KUKA KRL program: ps_b_etb_res_c03_R.src, ps_b_etb_res_c03_R.dat

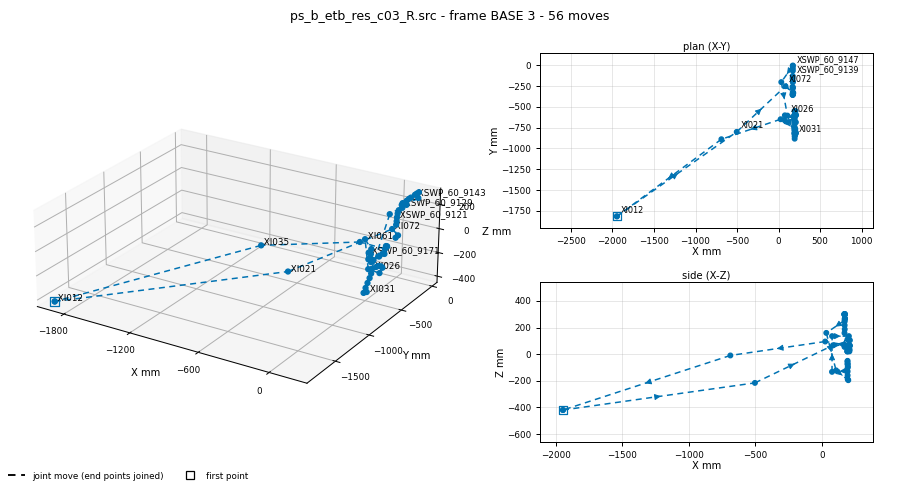
[picture p0: tool path of ps_b_etb_res_c03_R.src in frame BASE 3, 56 of 56 moves have a stored position in this frame; points joined in program order, loops and branches not executed]
--- ps_b_etb_res_c03_R.src ---
&ACCESS RVO2
&COMMENT Solda Atego STB
&PARAM DISKPATH = KRC:\R1\Program\olp
DEF ps_b_etb_res_c03_R( )
;FOLD INI
;FOLD SPOTTECH INI
USERSPOT(#INIT)
;ENDFOLD (SPOTTECH INI)
;FOLD GRIPPERTECH INI
USER_GRP(0,DUMMY,DUMMY,GDEFAULT)
;ENDFOLD (GRIPPERTECH INI)
  ;FOLD USER INI
    ;Make your modifications here

  ;ENDFOLD (USER INI)
;ENDFOLD (INI)

; Caraterizacao dos meios de producao
; Changes: Solda Respot - ATEGO STB
; Versao Atual: 30/03/2016
; Ferramenta: GUN C3
; Name: P13.050-R3
; optimised

chk_w5_wechs_ok ( )    ; CHECK GUN C3

if MaxStandMenge (3) then
 MaxStandmengeErreicht (3)
endif

IF (NOT(GHOST())) THEN
if Elektrodenwechsel ( 3 ) then
 e_fraes5 ()
endif
ENDIF

;FOLD PTP l012 Vel=100 % P_OLP37 Tool[5]:GUN C3 Base[3]:Atego/Axor;%{PE}%R 8.2.20,%MKUKATPBASIS,%CMOVE,%VPTP,%P 1:PTP, 2:l012, 3:, 5:100, 7:P_OLP37
$BWDSTART=FALSE
PDAT_ACT=PP_OLP37
FDAT_ACT=Fl012
BAS(#PTP_PARAMS,100)
PTP Xl012
;ENDFOLD

; AGUARDA LIBERACAO PARA SOLDAR RESPOT
;FOLD OUT 3333 'R3 trabalho concluído' State=FALSE ;%{PE}%R 8.2.20,%MKUKATPBASIS,%COUT,%VOUTX,%P 2:3333, 3:R3 trabalho concluído, 5:FALSE, 6:
$OUT[3333]=FALSE
;ENDFOLD
;FOLD OUT 3380 'Lib. p/ soldar Res Axor/Atego' State=TRUE ;%{PE}%R 8.2.20,%MKUKATPBASIS,%COUT,%VOUTX,%P 2:3380, 3:Lib. p/ soldar Res Axor/Atego, 5:TRUE, 6:
$OUT[3380]=TRUE
;ENDFOLD
;FOLD WAIT FOR ( IN 3380 'Lib. p/ soldar Res Axor/Atego' );%{PE}%R 8.2.20,%MKUKATPBASIS,%CEXT_WAIT_FOR,%VEXT_WAIT_FOR,%P 2:, 4:, 5:$IN, 6:3380, 7:Lib. p/ soldar Res Axor/Atego, 9:
WAIT FOR  ( $IN[3380] )
;ENDFOLD
;FOLD OUT 3380 'Lib. p/ soldar Res Axor/Atego' State=FALSE ;%{PE}%R 8.2.20,%MKUKATPBASIS,%COUT,%VOUTX,%P 2:3380, 3:Lib. p/ soldar Res Axor/Atego, 5:FALSE, 6:
$OUT[3380]=FALSE
;ENDFOLD
;FOLD OUT 3348 'Fora area GEOBOX' State=FALSE ;%{PE}%R 8.2.20,%MKUKATPBASIS,%COUT,%VOUTX,%P 2:3348, 3:Fora area GEOBOX, 5:FALSE, 6:
$OUT[3348]=FALSE
;ENDFOLD

;FOLD ; LIGA INTERTRAVAMENTO 4 SEGURANCA C/ GARRA DO R4;%{PE}%R 8.2.20,%MKUKATPBASIS,%CCOMMENT,%VNORMAL,%P 2:LIGA INTERTRAVAMENTO 4 SEGURANCA C/ GARRA DO R4
;ENDFOLD
;FOLD Collision.Monitoring_4_On ;%{PE}%MKUKATPUSER
COLLSTOP( 4, 1 ) ;Interrupt-Controlled
;ENDFOLD

;FOLD ; LIGA INTERTRAVAMENTO 13 COM R4 NA SOLDA;%{PE}%R 8.2.20,%MKUKATPBASIS,%CCOMMENT,%VNORMAL,%P 2:LIGA  INTERTRAVAMENTO  13  COM  R4  NA  SOLDA
;ENDFOLD
;FOLD Collision.Monitoring_AREA_7_On ;%{PE}%MKUKATPUSER
COLLSTOP( 13, 1 ) ;not Interrupt-Controlled
;ENDFOLD

;FOLD PTP l021 CONT Vel=100 % large Tool[5]:GUN C3 Base[3]:Atego/Axor;%{PE}%R 8.2.20,%MKUKATPBASIS,%CMOVE,%VPTP,%P 1:PTP, 2:l021, 3:C_DIS, 5:100, 7:large
$BWDSTART=FALSE
PDAT_ACT=Plarge
FDAT_ACT=Fl021
BAS(#PTP_PARAMS,100)
PTP Xl021 C_DIS
;ENDFOLD
;FOLD PTP l072 CONT Vel=100 % small Tool[5]:GUN C3 Base[3]:Atego/Axor;%{PE}%R 8.2.20,%MKUKATPBASIS,%CMOVE,%VPTP,%P 1:PTP, 2:l072, 3:C_DIS, 5:100, 7:small
$BWDSTART=FALSE
PDAT_ACT=Psmall
FDAT_ACT=Fl072
BAS(#PTP_PARAMS,100)
PTP Xl072 C_DIS
;ENDFOLD
;FOLD PTP l076 CONT Vel=100 % fin Tool[5]:GUN C3 Base[3]:Atego/Axor;%{PE}%R 8.2.20,%MKUKATPBASIS,%CMOVE,%VPTP,%P 1:PTP, 2:l076, 3:C_DIS, 5:100, 7:fin
$BWDSTART=FALSE
PDAT_ACT=Pfin
FDAT_ACT=Fl076
BAS(#PTP_PARAMS,100)
PTP Xl076 C_DIS
;ENDFOLD

;FOLD ; SWP_60_9103;%{PE}%R 8.2.20,%MKUKATPBASIS,%CCOMMENT,%VNORMAL,%P 2:SWP_60_9103
;ENDFOLD
;FOLD PTP SWP_60_9103 vmax SPOT Gun=3 RETR CLS PgNo1=200 ACTIVE=1 Tool[5]:GUN C3 Base[3]:Atego/Axor;%{PE}%R 8.2.2,%MKUKATPSPOT,%CSPOT,%VPTP,%P 1:PTP, 2:SWP_60_9103, 3:, 5:100, 7:vmax, 10:3, 12:#FIRST, 14:#CLO, 16:200, 18:1, 20:0, 22:0, 24:1, 25:NORMAL
$BWDSTART=FALSE
PDAT_ACT=Pvmax
FDAT_ACT=FSWP_60_9103
BAS(#PTP_PARAMS,Pvmax.VEL)
S_ACT.GUN=3
S_ACT.PAIR=SDEFAULT.PAIR
S_ACT.RETR=#CLO
S_ACT.CLO_TM=1
S_ACT.PGNO1=200
S_ACT.PGNO2=SDEFAULT.PGNO2
S_ACT.PRESS1=SDEFAULT.PRESS1
S_ACT.PRESS2=SDEFAULT.PRESS2
S_READY=FALSE
PTP XSWP_60_9103
USERSPOT(#SPOT, S_ACT)
WAIT FOR S_READY
;ENDFOLD

;FOLD ; SWP_60_9117;%{PE}%R 8.2.20,%MKUKATPBASIS,%CCOMMENT,%VNORMAL,%P 2:SWP_60_9117
;ENDFOLD
;FOLD PTP SWP_60_9117 vmax SPOT Gun=3 RETR CLS PgNo1=196 ACTIVE=1 Tool[5]:GUN C3 Base[3]:Atego/Axor;%{PE}%R 8.2.2,%MKUKATPSPOT,%CSPOT,%VPTP,%P 1:PTP, 2:SWP_60_9117, 3:, 5:100, 7:vmax, 10:3, 12:#FIRST, 14:#CLO, 16:196, 18:1, 20:0, 22:0, 24:1, 25:NORMAL
$BWDSTART=FALSE
PDAT_ACT=Pvmax
FDAT_ACT=FSWP_60_9117
BAS(#PTP_PARAMS,Pvmax.VEL)
S_ACT.GUN=3
S_ACT.PAIR=SDEFAULT.PAIR
S_ACT.RETR=#CLO
S_ACT.CLO_TM=1
S_ACT.PGNO1=196
S_ACT.PGNO2=SDEFAULT.PGNO2
S_ACT.PRESS1=SDEFAULT.PRESS1
S_ACT.PRESS2=SDEFAULT.PRESS2
S_READY=FALSE
PTP XSWP_60_9117
USERSPOT(#SPOT, S_ACT)
WAIT FOR S_READY
;ENDFOLD

;FOLD ; SWP_60_9119;%{PE}%R 8.2.20,%MKUKATPBASIS,%CCOMMENT,%VNORMAL,%P 2:SWP_60_9119
;ENDFOLD
;FOLD PTP SWP_60_9119 vmax SPOT Gun=3 RETR CLS PgNo1=196 ACTIVE=1 Tool[5]:GUN C3 Base[3]:Atego/Axor;%{PE}%R 8.2.2,%MKUKATPSPOT,%CSPOT,%VPTP,%P 1:PTP, 2:SWP_60_9119, 3:, 5:100, 7:vmax, 10:3, 12:#FIRST, 14:#CLO, 16:196, 18:1, 20:0, 22:0, 24:1, 25:NORMAL
$BWDSTART=FALSE
PDAT_ACT=Pvmax
FDAT_ACT=FSWP_60_9119
BAS(#PTP_PARAMS,Pvmax.VEL)
S_ACT.GUN=3
S_ACT.PAIR=SDEFAULT.PAIR
S_ACT.RETR=#CLO
S_ACT.CLO_TM=1
S_ACT.PGNO1=196
S_ACT.PGNO2=SDEFAULT.PGNO2
S_ACT.PRESS1=SDEFAULT.PRESS1
S_ACT.PRESS2=SDEFAULT.PRESS2
S_READY=FALSE
PTP XSWP_60_9119
USERSPOT(#SPOT, S_ACT)
WAIT FOR S_READY
;ENDFOLD

;FOLD ; SWP_60_9121;%{PE}%R 8.2.20,%MKUKATPBASIS,%CCOMMENT,%VNORMAL,%P 2:SWP_60_9121
;ENDFOLD
;FOLD PTP SWP_60_9121 vmax SPOT Gun=3 RETR CLS PgNo1=196 ACTIVE=1 Tool[5]:GUN C3 Base[3]:Atego/Axor;%{PE}%R 8.2.2,%MKUKATPSPOT,%CSPOT,%VPTP,%P 1:PTP, 2:SWP_60_9121, 3:, 5:100, 7:vmax, 10:3, 12:#FIRST, 14:#CLO, 16:196, 18:1, 20:0, 22:0, 24:1, 25:NORMAL
$BWDSTART=FALSE
PDAT_ACT=Pvmax
FDAT_ACT=FSWP_60_9121
BAS(#PTP_PARAMS,Pvmax.VEL)
S_ACT.GUN=3
S_ACT.PAIR=SDEFAULT.PAIR
S_ACT.RETR=#CLO
S_ACT.CLO_TM=1
S_ACT.PGNO1=196
S_ACT.PGNO2=SDEFAULT.PGNO2
S_ACT.PRESS1=SDEFAULT.PRESS1
S_ACT.PRESS2=SDEFAULT.PRESS2
S_READY=FALSE
PTP XSWP_60_9121
USERSPOT(#SPOT, S_ACT)
WAIT FOR S_READY
;ENDFOLD

;FOLD ; SWP_60_9123;%{PE}%R 8.2.20,%MKUKATPBASIS,%CCOMMENT,%VNORMAL,%P 2:SWP_60_9123
;ENDFOLD
;FOLD PTP SWP_60_9123 vmax SPOT Gun=3 RETR CLS PgNo1=196 ACTIVE=1 Tool[5]:GUN C3 Base[3]:Atego/Axor;%{PE}%R 8.2.2,%MKUKATPSPOT,%CSPOT,%VPTP,%P 1:PTP, 2:SWP_60_9123, 3:, 5:100, 7:vmax, 10:3, 12:#FIRST, 14:#CLO, 16:196, 18:1, 20:0, 22:0, 24:1, 25:NORMAL
$BWDSTART=FALSE
PDAT_ACT=Pvmax
FDAT_ACT=FSWP_60_9123
BAS(#PTP_PARAMS,Pvmax.VEL)
S_ACT.GUN=3
S_ACT.PAIR=SDEFAULT.PAIR
S_ACT.RETR=#CLO
S_ACT.CLO_TM=1
S_ACT.PGNO1=196
S_ACT.PGNO2=SDEFAULT.PGNO2
S_ACT.PRESS1=SDEFAULT.PRESS1
S_ACT.PRESS2=SDEFAULT.PRESS2
S_READY=FALSE
PTP XSWP_60_9123
USERSPOT(#SPOT, S_ACT)
WAIT FOR S_READY
;ENDFOLD

;FOLD ; SWP_60_9125;%{PE}%R 8.2.20,%MKUKATPBASIS,%CCOMMENT,%VNORMAL,%P 2:SWP_60_9125
;ENDFOLD
;FOLD PTP SWP_60_9125 vmax SPOT Gun=3 RETR CLS PgNo1=196 ACTIVE=1 Tool[5]:GUN C3 Base[3]:Atego/Axor;%{PE}%R 8.2.2,%MKUKATPSPOT,%CSPOT,%VPTP,%P 1:PTP, 2:SWP_60_9125, 3:, 5:100, 7:vmax, 10:3, 12:#FIRST, 14:#CLO, 16:196, 18:1, 20:0, 22:0, 24:1, 25:NORMAL
$BWDSTART=FALSE
PDAT_ACT=Pvmax
FDAT_ACT=FSWP_60_9125
BAS(#PTP_PARAMS,Pvmax.VEL)
S_ACT.GUN=3
S_ACT.PAIR=SDEFAULT.PAIR
S_ACT.RETR=#CLO
S_ACT.CLO_TM=1
S_ACT.PGNO1=196
S_ACT.PGNO2=SDEFAULT.PGNO2
S_ACT.PRESS1=SDEFAULT.PRESS1
S_ACT.PRESS2=SDEFAULT.PRESS2
S_READY=FALSE
PTP XSWP_60_9125
USERSPOT(#SPOT, S_ACT)
WAIT FOR S_READY
;ENDFOLD

;FOLD ; SWP_60_9129;%{PE}%R 8.2.20,%MKUKATPBASIS,%CCOMMENT,%VNORMAL,%P 2:SWP_60_9129
;ENDFOLD
;FOLD PTP SWP_60_9129 vmax SPOT Gun=3 RETR CLS PgNo1=196 ACTIVE=1 Tool[5]:GUN C3 Base[3]:Atego/Axor;%{PE}%R 8.2.2,%MKUKATPSPOT,%CSPOT,%VPTP,%P 1:PTP, 2:SWP_60_9129, 3:, 5:100, 7:vmax, 10:3, 12:#FIRST, 14:#CLO, 16:196, 18:1, 20:0, 22:0, 24:1, 25:NORMAL
$BWDSTART=FALSE
PDAT_ACT=Pvmax
FDAT_ACT=FSWP_60_9129
BAS(#PTP_PARAMS,Pvmax.VEL)
S_ACT.GUN=3
S_ACT.PAIR=SDEFAULT.PAIR
S_ACT.RETR=#CLO
S_ACT.CLO_TM=1
S_ACT.PGNO1=196
S_ACT.PGNO2=SDEFAULT.PGNO2
S_ACT.PRESS1=SDEFAULT.PRESS1
S_ACT.PRESS2=SDEFAULT.PRESS2
S_READY=FALSE
PTP XSWP_60_9129
USERSPOT(#SPOT, S_ACT)
WAIT FOR S_READY
;ENDFOLD

;FOLD ; SWP_60_9131;%{PE}%R 8.2.20,%MKUKATPBASIS,%CCOMMENT,%VNORMAL,%P 2:SWP_60_9131
;ENDFOLD
;FOLD PTP SWP_60_9131 vmax SPOT Gun=3 RETR CLS PgNo1=196 ACTIVE=1 Tool[5]:GUN C3 Base[3]:Atego/Axor;%{PE}%R 8.2.2,%MKUKATPSPOT,%CSPOT,%VPTP,%P 1:PTP, 2:SWP_60_9131, 3:, 5:100, 7:vmax, 10:3, 12:#FIRST, 14:#CLO, 16:196, 18:1, 20:0, 22:0, 24:1, 25:NORMAL
$BWDSTART=FALSE
PDAT_ACT=Pvmax
FDAT_ACT=FSWP_60_9131
BAS(#PTP_PARAMS,Pvmax.VEL)
S_ACT.GUN=3
S_ACT.PAIR=SDEFAULT.PAIR
S_ACT.RETR=#CLO
S_ACT.CLO_TM=1
S_ACT.PGNO1=196
S_ACT.PGNO2=SDEFAULT.PGNO2
S_ACT.PRESS1=SDEFAULT.PRESS1
S_ACT.PRESS2=SDEFAULT.PRESS2
S_READY=FALSE
PTP XSWP_60_9131
USERSPOT(#SPOT, S_ACT)
WAIT FOR S_READY
;ENDFOLD

;FOLD PTP l077 CONT Vel=100 % fin Tool[5]:GUN C3 Base[3]:Atego/Axor;%{PE}%R 8.2.20,%MKUKATPBASIS,%CMOVE,%VPTP,%P 1:PTP, 2:l077, 3:C_DIS, 5:100, 7:fin
$BWDSTART=FALSE
PDAT_ACT=Pfin
FDAT_ACT=Fl077
BAS(#PTP_PARAMS,100)
PTP Xl077 C_DIS
;ENDFOLD
;FOLD PTP l078 CONT Vel=100 % fin Tool[5]:GUN C3 Base[3]:Atego/Axor;%{PE}%R 8.2.20,%MKUKATPBASIS,%CMOVE,%VPTP,%P 1:PTP, 2:l078, 3:C_DIS, 5:100, 7:fin
$BWDSTART=FALSE
PDAT_ACT=Pfin
FDAT_ACT=Fl078
BAS(#PTP_PARAMS,100)
PTP Xl078 C_DIS
;ENDFOLD

;FOLD ; SWP_60_9135;%{PE}%R 8.2.20,%MKUKATPBASIS,%CCOMMENT,%VNORMAL,%P 2:SWP_60_9135
;ENDFOLD
;FOLD PTP SWP_60_9135 vmax SPOT Gun=3 RETR CLS PgNo1=196 ACTIVE=1 Tool[5]:GUN C3 Base[3]:Atego/Axor;%{PE}%R 8.2.2,%MKUKATPSPOT,%CSPOT,%VPTP,%P 1:PTP, 2:SWP_60_9135, 3:, 5:100, 7:vmax, 10:3, 12:#FIRST, 14:#CLO, 16:196, 18:1, 20:0, 22:0, 24:1, 25:NORMAL
$BWDSTART=FALSE
PDAT_ACT=Pvmax
FDAT_ACT=FSWP_60_9135
BAS(#PTP_PARAMS,Pvmax.VEL)
S_ACT.GUN=3
S_ACT.PAIR=SDEFAULT.PAIR
S_ACT.RETR=#CLO
S_ACT.CLO_TM=1
S_ACT.PGNO1=196
S_ACT.PGNO2=SDEFAULT.PGNO2
S_ACT.PRESS1=SDEFAULT.PRESS1
S_ACT.PRESS2=SDEFAULT.PRESS2
S_READY=FALSE
PTP XSWP_60_9135
USERSPOT(#SPOT, S_ACT)
WAIT FOR S_READY
;ENDFOLD

;FOLD ; SWP_60_9137;%{PE}%R 8.2.20,%MKUKATPBASIS,%CCOMMENT,%VNORMAL,%P 2:SWP_60_9137
;ENDFOLD
;FOLD PTP SWP_60_9137 vmax SPOT Gun=3 RETR CLS PgNo1=196 ACTIVE=1 Tool[5]:GUN C3 Base[3]:Atego/Axor;%{PE}%R 8.2.2,%MKUKATPSPOT,%CSPOT,%VPTP,%P 1:PTP, 2:SWP_60_9137, 3:, 5:100, 7:vmax, 10:3, 12:#FIRST, 14:#CLO, 16:196, 18:1, 20:0, 22:0, 24:1, 25:NORMAL
$BWDSTART=FALSE
PDAT_ACT=Pvmax
FDAT_ACT=FSWP_60_9137
BAS(#PTP_PARAMS,Pvmax.VEL)
S_ACT.GUN=3
S_ACT.PAIR=SDEFAULT.PAIR
S_ACT.RETR=#CLO
S_ACT.CLO_TM=1
S_ACT.PGNO1=196
S_ACT.PGNO2=SDEFAULT.PGNO2
S_ACT.PRESS1=SDEFAULT.PRESS1
S_ACT.PRESS2=SDEFAULT.PRESS2
S_READY=FALSE
PTP XSWP_60_9137
USERSPOT(#SPOT, S_ACT)
WAIT FOR S_READY
;ENDFOLD

;FOLD ; SWP_60_9139;%{PE}%R 8.2.20,%MKUKATPBASIS,%CCOMMENT,%VNORMAL,%P 2:SWP_60_9139
;ENDFOLD
;FOLD PTP SWP_60_9139 vmax SPOT Gun=3 RETR CLS PgNo1=196 ACTIVE=1 Tool[5]:GUN C3 Base[3]:Atego/Axor;%{PE}%R 8.2.2,%MKUKATPSPOT,%CSPOT,%VPTP,%P 1:PTP, 2:SWP_60_9139, 3:, 5:100, 7:vmax, 10:3, 12:#FIRST, 14:#CLO, 16:196, 18:1, 20:0, 22:0, 24:1, 25:NORMAL
$BWDSTART=FALSE
PDAT_ACT=Pvmax
FDAT_ACT=FSWP_60_9139
BAS(#PTP_PARAMS,Pvmax.VEL)
S_ACT.GUN=3
S_ACT.PAIR=SDEFAULT.PAIR
S_ACT.RETR=#CLO
S_ACT.CLO_TM=1
S_ACT.PGNO1=196
S_ACT.PGNO2=SDEFAULT.PGNO2
S_ACT.PRESS1=SDEFAULT.PRESS1
S_ACT.PRESS2=SDEFAULT.PRESS2
S_READY=FALSE
PTP XSWP_60_9139
USERSPOT(#SPOT, S_ACT)
WAIT FOR S_READY
;ENDFOLD

;FOLD ; SWP_60_9143;%{PE}%R 8.2.20,%MKUKATPBASIS,%CCOMMENT,%VNORMAL,%P 2:SWP_60_9143
;ENDFOLD
;FOLD PTP SWP_60_9143 vmax SPOT Gun=3 RETR CLS PgNo1=196 ACTIVE=1 Tool[5]:GUN C3 Base[3]:Atego/Axor;%{PE}%R 8.2.2,%MKUKATPSPOT,%CSPOT,%VPTP,%P 1:PTP, 2:SWP_60_9143, 3:, 5:100, 7:vmax, 10:3, 12:#FIRST, 14:#CLO, 16:196, 18:1, 20:0, 22:0, 24:1, 25:NORMAL
$BWDSTART=FALSE
PDAT_ACT=Pvmax
FDAT_ACT=FSWP_60_9143
BAS(#PTP_PARAMS,Pvmax.VEL)
S_ACT.GUN=3
S_ACT.PAIR=SDEFAULT.PAIR
S_ACT.RETR=#CLO
S_ACT.CLO_TM=1
S_ACT.PGNO1=196
S_ACT.PGNO2=SDEFAULT.PGNO2
S_ACT.PRESS1=SDEFAULT.PRESS1
S_ACT.PRESS2=SDEFAULT.PRESS2
S_READY=FALSE
PTP XSWP_60_9143
USERSPOT(#SPOT, S_ACT)
WAIT FOR S_READY
;ENDFOLD

;FOLD ; SWP_60_9145;%{PE}%R 8.2.20,%MKUKATPBASIS,%CCOMMENT,%VNORMAL,%P 2:SWP_60_9145
;ENDFOLD
;FOLD PTP SWP_60_9145 vmax SPOT Gun=3 RETR CLS PgNo1=196 ACTIVE=1 Tool[5]:GUN C3 Base[3]:Atego/Axor;%{PE}%R 8.2.2,%MKUKATPSPOT,%CSPOT,%VPTP,%P 1:PTP, 2:SWP_60_9145, 3:, 5:100, 7:vmax, 10:3, 12:#FIRST, 14:#CLO, 16:196, 18:1, 20:0, 22:0, 24:1, 25:NORMAL
$BWDSTART=FALSE
PDAT_ACT=Pvmax
FDAT_ACT=FSWP_60_9145
BAS(#PTP_PARAMS,Pvmax.VEL)
S_ACT.GUN=3
S_ACT.PAIR=SDEFAULT.PAIR
S_ACT.RETR=#CLO
S_ACT.CLO_TM=1
S_ACT.PGNO1=196
S_ACT.PGNO2=SDEFAULT.PGNO2
S_ACT.PRESS1=SDEFAULT.PRESS1
S_ACT.PRESS2=SDEFAULT.PRESS2
S_READY=FALSE
PTP XSWP_60_9145
USERSPOT(#SPOT, S_ACT)
WAIT FOR S_READY
;ENDFOLD

;FOLD ; SWP_60_9147;%{PE}%R 8.2.20,%MKUKATPBASIS,%CCOMMENT,%VNORMAL,%P 2:SWP_60_9147
;ENDFOLD
;FOLD PTP SWP_60_9147 vmax SPOT Gun=3 RETR CLS PgNo1=196 ACTIVE=1 Tool[5]:GUN C3 Base[3]:Atego/Axor;%{PE}%R 8.2.2,%MKUKATPSPOT,%CSPOT,%VPTP,%P 1:PTP, 2:SWP_60_9147, 3:, 5:100, 7:vmax, 10:3, 12:#FIRST, 14:#CLO, 16:196, 18:1, 20:0, 22:0, 24:1, 25:NORMAL
$BWDSTART=FALSE
PDAT_ACT=Pvmax
FDAT_ACT=FSWP_60_9147
BAS(#PTP_PARAMS,Pvmax.VEL)
S_ACT.GUN=3
S_ACT.PAIR=SDEFAULT.PAIR
S_ACT.RETR=#CLO
S_ACT.CLO_TM=1
S_ACT.PGNO1=196
S_ACT.PGNO2=SDEFAULT.PGNO2
S_ACT.PRESS1=SDEFAULT.PRESS1
S_ACT.PRESS2=SDEFAULT.PRESS2
S_READY=FALSE
PTP XSWP_60_9147
USERSPOT(#SPOT, S_ACT)
WAIT FOR S_READY
;ENDFOLD

;FOLD PTP l116 CONT Vel=100 % small Tool[5]:GUN C3 Base[3]:Atego/Axor;%{PE}%R 8.2.20,%MKUKATPBASIS,%CMOVE,%VPTP,%P 1:PTP, 2:l116, 3:C_DIS, 5:100, 7:small
$BWDSTART=FALSE
PDAT_ACT=Psmall
FDAT_ACT=Fl116
BAS(#PTP_PARAMS,100)
PTP Xl116 C_DIS
;ENDFOLD
;FOLD PTP l044 CONT Vel=100 % large Tool[5]:GUN C3 Base[3]:Atego/Axor;%{PE}%R 8.2.20,%MKUKATPBASIS,%CMOVE,%VPTP,%P 1:PTP, 2:l044, 3:C_DIS, 5:100, 7:large
$BWDSTART=FALSE
PDAT_ACT=Plarge
FDAT_ACT=Fl044
BAS(#PTP_PARAMS,100)
PTP Xl044 C_DIS
;ENDFOLD
;FOLD PTP l026 CONT Vel=100 % large Tool[5]:GUN C3 Base[3]:Atego/Axor;%{PE}%R 8.2.20,%MKUKATPBASIS,%CMOVE,%VPTP,%P 1:PTP, 2:l026, 3:C_DIS, 5:100, 7:large
$BWDSTART=FALSE
PDAT_ACT=Plarge
FDAT_ACT=Fl026
BAS(#PTP_PARAMS,100)
PTP Xl026 C_DIS
;ENDFOLD
;FOLD PTP l031 CONT Vel=100 % fin Tool[5]:GUN C3 Base[3]:Atego/Axor;%{PE}%R 8.2.20,%MKUKATPBASIS,%CMOVE,%VPTP,%P 1:PTP, 2:l031, 3:C_DIS, 5:100, 7:fin
$BWDSTART=FALSE
PDAT_ACT=Pfin
FDAT_ACT=Fl031
BAS(#PTP_PARAMS,100)
PTP Xl031 C_DIS
;ENDFOLD

;FOLD ; SWP_60_9041;%{PE}%R 8.2.20,%MKUKATPBASIS,%CCOMMENT,%VNORMAL,%P 2:SWP_60_9041
;ENDFOLD
;FOLD PTP SWP_60_9041 vmax SPOT Gun=3 RETR CLS PgNo1=196 ACTIVE=1 Tool[5]:GUN C3 Base[3]:Atego/Axor;%{PE}%R 8.2.2,%MKUKATPSPOT,%CSPOT,%VPTP,%P 1:PTP, 2:SWP_60_9041, 3:, 5:100, 7:vmax, 10:3, 12:#FIRST, 14:#CLO, 16:196, 18:1, 20:0, 22:0, 24:1, 25:NORMAL
$BWDSTART=FALSE
PDAT_ACT=Pvmax
FDAT_ACT=FSWP_60_9041
BAS(#PTP_PARAMS,Pvmax.VEL)
S_ACT.GUN=3
S_ACT.PAIR=SDEFAULT.PAIR
S_ACT.RETR=#CLO
S_ACT.CLO_TM=1
S_ACT.PGNO1=196
S_ACT.PGNO2=SDEFAULT.PGNO2
S_ACT.PRESS1=SDEFAULT.PRESS1
S_ACT.PRESS2=SDEFAULT.PRESS2
S_READY=FALSE
PTP XSWP_60_9041
USERSPOT(#SPOT, S_ACT)
WAIT FOR S_READY
;ENDFOLD

;FOLD ; DESLIGA INTERTRAVAMENTO 13 COM R4 NA SOLDA;%{PE}%R 8.2.20,%MKUKATPBASIS,%CCOMMENT,%VNORMAL,%P 2:DESLIGA  INTERTRAVAMENTO  13  COM  R4  NA  SOLDA
;ENDFOLD
;FOLD Collision.Monitoring_AREA_7_Off . ;%{PE}%MKUKATPUSER
COLLSTOP( 13, 2+0 )
;ENDFOLD

;FOLD ; SWP_60_9039;%{PE}%R 8.2.20,%MKUKATPBASIS,%CCOMMENT,%VNORMAL,%P 2:SWP_60_9039
;ENDFOLD
;FOLD PTP SWP_60_9039 vmax SPOT Gun=3 RETR CLS PgNo1=196 ACTIVE=1 Tool[5]:GUN C3 Base[3]:Atego/Axor;%{PE}%R 8.2.2,%MKUKATPSPOT,%CSPOT,%VPTP,%P 1:PTP, 2:SWP_60_9039, 3:, 5:100, 7:vmax, 10:3, 12:#FIRST, 14:#CLO, 16:196, 18:1, 20:0, 22:0, 24:1, 25:NORMAL
$BWDSTART=FALSE
PDAT_ACT=Pvmax
FDAT_ACT=FSWP_60_9039
BAS(#PTP_PARAMS,Pvmax.VEL)
S_ACT.GUN=3
S_ACT.PAIR=SDEFAULT.PAIR
S_ACT.RETR=#CLO
S_ACT.CLO_TM=1
S_ACT.PGNO1=196
S_ACT.PGNO2=SDEFAULT.PGNO2
S_ACT.PRESS1=SDEFAULT.PRESS1
S_ACT.PRESS2=SDEFAULT.PRESS2
S_READY=FALSE
PTP XSWP_60_9039
USERSPOT(#SPOT, S_ACT)
WAIT FOR S_READY
;ENDFOLD

;FOLD ; SWP_60_9037;%{PE}%R 8.2.20,%MKUKATPBASIS,%CCOMMENT,%VNORMAL,%P 2:SWP_60_9037
;ENDFOLD
;FOLD PTP SWP_60_9037 vmax SPOT Gun=3 RETR CLS PgNo1=196 ACTIVE=1 Tool[5]:GUN C3 Base[3]:Atego/Axor;%{PE}%R 8.2.2,%MKUKATPSPOT,%CSPOT,%VPTP,%P 1:PTP, 2:SWP_60_9037, 3:, 5:100, 7:vmax, 10:3, 12:#FIRST, 14:#CLO, 16:196, 18:1, 20:0, 22:0, 24:1, 25:NORMAL
$BWDSTART=FALSE
PDAT_ACT=Pvmax
FDAT_ACT=FSWP_60_9037
BAS(#PTP_PARAMS,Pvmax.VEL)
S_ACT.GUN=3
S_ACT.PAIR=SDEFAULT.PAIR
S_ACT.RETR=#CLO
S_ACT.CLO_TM=1
S_ACT.PGNO1=196
S_ACT.PGNO2=SDEFAULT.PGNO2
S_ACT.PRESS1=SDEFAULT.PRESS1
S_ACT.PRESS2=SDEFAULT.PRESS2
S_READY=FALSE
PTP XSWP_60_9037
USERSPOT(#SPOT, S_ACT)
WAIT FOR S_READY
;ENDFOLD

;FOLD ; SWP_60_9035;%{PE}%R 8.2.20,%MKUKATPBASIS,%CCOMMENT,%VNORMAL,%P 2:SWP_60_9035
;ENDFOLD
;FOLD PTP SWP_60_9035 vmax SPOT Gun=3 RETR CLS PgNo1=196 ACTIVE=1 Tool[5]:GUN C3 Base[3]:Atego/Axor;%{PE}%R 8.2.2,%MKUKATPSPOT,%CSPOT,%VPTP,%P 1:PTP, 2:SWP_60_9035, 3:, 5:100, 7:vmax, 10:3, 12:#FIRST, 14:#CLO, 16:196, 18:1, 20:0, 22:0, 24:1, 25:NORMAL
$BWDSTART=FALSE
PDAT_ACT=Pvmax
FDAT_ACT=FSWP_60_9035
BAS(#PTP_PARAMS,Pvmax.VEL)
S_ACT.GUN=3
S_ACT.PAIR=SDEFAULT.PAIR
S_ACT.RETR=#CLO
S_ACT.CLO_TM=1
S_ACT.PGNO1=196
S_ACT.PGNO2=SDEFAULT.PGNO2
S_ACT.PRESS1=SDEFAULT.PRESS1
S_ACT.PRESS2=SDEFAULT.PRESS2
S_READY=FALSE
PTP XSWP_60_9035
USERSPOT(#SPOT, S_ACT)
WAIT FOR S_READY
;ENDFOLD

;FOLD ; SWP_60_9033;%{PE}%R 8.2.20,%MKUKATPBASIS,%CCOMMENT,%VNORMAL,%P 2:SWP_60_9033
;ENDFOLD
;FOLD PTP SWP_60_9033 vmax SPOT Gun=3 RETR CLS PgNo1=196 ACTIVE=1 Tool[5]:GUN C3 Base[3]:Atego/Axor;%{PE}%R 8.2.2,%MKUKATPSPOT,%CSPOT,%VPTP,%P 1:PTP, 2:SWP_60_9033, 3:, 5:100, 7:vmax, 10:3, 12:#FIRST, 14:#CLO, 16:196, 18:1, 20:0, 22:0, 24:1, 25:NORMAL
$BWDSTART=FALSE
PDAT_ACT=Pvmax
FDAT_ACT=FSWP_60_9033
BAS(#PTP_PARAMS,Pvmax.VEL)
S_ACT.GUN=3
S_ACT.PAIR=SDEFAULT.PAIR
S_ACT.RETR=#CLO
S_ACT.CLO_TM=1
S_ACT.PGNO1=196
S_ACT.PGNO2=SDEFAULT.PGNO2
S_ACT.PRESS1=SDEFAULT.PRESS1
S_ACT.PRESS2=SDEFAULT.PRESS2
S_READY=FALSE
PTP XSWP_60_9033
USERSPOT(#SPOT, S_ACT)
WAIT FOR S_READY
;ENDFOLD

;FOLD ; SWP_60_9029;%{PE}%R 8.2.20,%MKUKATPBASIS,%CCOMMENT,%VNORMAL,%P 2:SWP_60_9029
;ENDFOLD
;FOLD PTP SWP_60_9029 vmax SPOT Gun=3 RETR CLS PgNo1=196 ACTIVE=1 Tool[5]:GUN C3 Base[3]:Atego/Axor;%{PE}%R 8.2.2,%MKUKATPSPOT,%CSPOT,%VPTP,%P 1:PTP, 2:SWP_60_9029, 3:, 5:100, 7:vmax, 10:3, 12:#FIRST, 14:#CLO, 16:196, 18:1, 20:0, 22:0, 24:1, 25:NORMAL
$BWDSTART=FALSE
PDAT_ACT=Pvmax
FDAT_ACT=FSWP_60_9029
BAS(#PTP_PARAMS,Pvmax.VEL)
S_ACT.GUN=3
S_ACT.PAIR=SDEFAULT.PAIR
S_ACT.RETR=#CLO
S_ACT.CLO_TM=1
S_ACT.PGNO1=196
S_ACT.PGNO2=SDEFAULT.PGNO2
S_ACT.PRESS1=SDEFAULT.PRESS1
S_ACT.PRESS2=SDEFAULT.PRESS2
S_READY=FALSE
PTP XSWP_60_9029
USERSPOT(#SPOT, S_ACT)
WAIT FOR S_READY
;ENDFOLD

;FOLD ; SWP_60_9027;%{PE}%R 8.2.20,%MKUKATPBASIS,%CCOMMENT,%VNORMAL,%P 2:SWP_60_9027
;ENDFOLD
;FOLD PTP SWP_60_9027 vmax SPOT Gun=3 RETR CLS PgNo1=196 ACTIVE=1 Tool[5]:GUN C3 Base[3]:Atego/Axor;%{PE}%R 8.2.2,%MKUKATPSPOT,%CSPOT,%VPTP,%P 1:PTP, 2:SWP_60_9027, 3:, 5:100, 7:vmax, 10:3, 12:#FIRST, 14:#CLO, 16:196, 18:1, 20:0, 22:0, 24:1, 25:NORMAL
$BWDSTART=FALSE
PDAT_ACT=Pvmax
FDAT_ACT=FSWP_60_9027
BAS(#PTP_PARAMS,Pvmax.VEL)
S_ACT.GUN=3
S_ACT.PAIR=SDEFAULT.PAIR
S_ACT.RETR=#CLO
S_ACT.CLO_TM=1
S_ACT.PGNO1=196
S_ACT.PGNO2=SDEFAULT.PGNO2
S_ACT.PRESS1=SDEFAULT.PRESS1
S_ACT.PRESS2=SDEFAULT.PRESS2
S_READY=FALSE
PTP XSWP_60_9027
USERSPOT(#SPOT, S_ACT)
WAIT FOR S_READY
;ENDFOLD

;FOLD ; SWP_60_9025;%{PE}%R 8.2.20,%MKUKATPBASIS,%CCOMMENT,%VNORMAL,%P 2:SWP_60_9025
;ENDFOLD
;FOLD PTP SWP_60_9025 vmax SPOT Gun=3 RETR CLS PgNo1=200 ACTIVE=1 Tool[5]:GUN C3 Base[3]:Atego/Axor;%{PE}%R 8.2.2,%MKUKATPSPOT,%CSPOT,%VPTP,%P 1:PTP, 2:SWP_60_9025, 3:, 5:100, 7:vmax, 10:3, 12:#FIRST, 14:#CLO, 16:200, 18:1, 20:0, 22:0, 24:1, 25:NORMAL
$BWDSTART=FALSE
PDAT_ACT=Pvmax
FDAT_ACT=FSWP_60_9025
BAS(#PTP_PARAMS,Pvmax.VEL)
S_ACT.GUN=3
S_ACT.PAIR=SDEFAULT.PAIR
S_ACT.RETR=#CLO
S_ACT.CLO_TM=1
S_ACT.PGNO1=200
S_ACT.PGNO2=SDEFAULT.PGNO2
S_ACT.PRESS1=SDEFAULT.PRESS1
S_ACT.PRESS2=SDEFAULT.PRESS2
S_READY=FALSE
PTP XSWP_60_9025
USERSPOT(#SPOT, S_ACT)
WAIT FOR S_READY
;ENDFOLD

;FOLD ; SWP_60_9023;%{PE}%R 8.2.20,%MKUKATPBASIS,%CCOMMENT,%VNORMAL,%P 2:SWP_60_9023
;ENDFOLD
;FOLD PTP SWP_60_9023 vmax SPOT Gun=3 RETR CLS PgNo1=200 ACTIVE=1 Tool[5]:GUN C3 Base[3]:Atego/Axor;%{PE}%R 8.2.2,%MKUKATPSPOT,%CSPOT,%VPTP,%P 1:PTP, 2:SWP_60_9023, 3:, 5:100, 7:vmax, 10:3, 12:#FIRST, 14:#CLO, 16:200, 18:1, 20:0, 22:0, 24:1, 25:NORMAL
$BWDSTART=FALSE
PDAT_ACT=Pvmax
FDAT_ACT=FSWP_60_9023
BAS(#PTP_PARAMS,Pvmax.VEL)
S_ACT.GUN=3
S_ACT.PAIR=SDEFAULT.PAIR
S_ACT.RETR=#CLO
S_ACT.CLO_TM=1
S_ACT.PGNO1=200
S_ACT.PGNO2=SDEFAULT.PGNO2
S_ACT.PRESS1=SDEFAULT.PRESS1
S_ACT.PRESS2=SDEFAULT.PRESS2
S_READY=FALSE
PTP XSWP_60_9023
USERSPOT(#SPOT, S_ACT)
WAIT FOR S_READY
;ENDFOLD

;FOLD PTP l055 CONT Vel=100 % fin Tool[5]:GUN C3 Base[3]:Atego/Axor;%{PE}%R 8.2.20,%MKUKATPBASIS,%CMOVE,%VPTP,%P 1:PTP, 2:l055, 3:C_DIS, 5:100, 7:fin
$BWDSTART=FALSE
PDAT_ACT=Pfin
FDAT_ACT=Fl055
BAS(#PTP_PARAMS,100)
PTP Xl055 C_DIS
;ENDFOLD
;FOLD PTP l060 CONT Vel=100 % large Tool[5]:GUN C3 Base[3]:Atego/Axor;%{PE}%R 8.2.20,%MKUKATPBASIS,%CMOVE,%VPTP,%P 1:PTP, 2:l060, 3:C_DIS, 5:100, 7:large
$BWDSTART=FALSE
PDAT_ACT=Plarge
FDAT_ACT=Fl060
BAS(#PTP_PARAMS,100)
PTP Xl060 C_DIS
;ENDFOLD
;FOLD PTP l061 CONT Vel=100 % medium Tool[5]:GUN C3 Base[3]:Atego/Axor;%{PE}%R 8.2.20,%MKUKATPBASIS,%CMOVE,%VPTP,%P 1:PTP, 2:l061, 3:C_DIS, 5:100, 7:medium
$BWDSTART=FALSE
PDAT_ACT=Pmedium
FDAT_ACT=Fl061
BAS(#PTP_PARAMS,100)
PTP Xl061 C_DIS
;ENDFOLD
;FOLD PTP l062 CONT Vel=100 % fin Tool[5]:GUN C3 Base[3]:Atego/Axor;%{PE}%R 8.2.20,%MKUKATPBASIS,%CMOVE,%VPTP,%P 1:PTP, 2:l062, 3:C_DIS, 5:100, 7:fin
$BWDSTART=FALSE
PDAT_ACT=Pfin
FDAT_ACT=Fl062
BAS(#PTP_PARAMS,100)
PTP Xl062 C_DIS
;ENDFOLD

;FOLD ; Inicio dos Pontos adiconados;%{PE}%R 8.2.20,%MKUKATPBASIS,%CCOMMENT,%VNORMAL,%P 2:Inicio  dos  Pontos adiconados
;ENDFOLD

;FOLD ; SWP_60_9171;%{PE}%R 8.2.20,%MKUKATPBASIS,%CCOMMENT,%VNORMAL,%P 2:SWP_60_9171
;ENDFOLD
;FOLD PTP SWP_60_9171 vmax SPOT Gun=3 RETR CLS PgNo1=201 ACTIVE=1 Tool[5]:GUN C3 Base[3]:Atego/Axor;%{PE}%R 8.2.2,%MKUKATPSPOT,%CSPOT,%VPTP,%P 1:PTP, 2:SWP_60_9171, 3:, 5:100, 7:vmax, 10:3, 12:#FIRST, 14:#CLO, 16:201, 18:1, 20:0, 22:0, 24:1, 25:NORMAL
$BWDSTART=FALSE
PDAT_ACT=Pvmax
FDAT_ACT=FSWP_60_9171
BAS(#PTP_PARAMS,Pvmax.VEL)
S_ACT.GUN=3
S_ACT.PAIR=SDEFAULT.PAIR
S_ACT.RETR=#CLO
S_ACT.CLO_TM=1
S_ACT.PGNO1=201
S_ACT.PGNO2=SDEFAULT.PGNO2
S_ACT.PRESS1=SDEFAULT.PRESS1
S_ACT.PRESS2=SDEFAULT.PRESS2
S_READY=FALSE
PTP XSWP_60_9171
USERSPOT(#SPOT, S_ACT)
WAIT FOR S_READY
;ENDFOLD

;FOLD PTP l064 CONT Vel=100 % fin Tool[5]:GUN C3 Base[3]:Atego/Axor;%{PE}%R 8.2.20,%MKUKATPBASIS,%CMOVE,%VPTP,%P 1:PTP, 2:l064, 3:C_DIS, 5:100, 7:fin
$BWDSTART=FALSE
PDAT_ACT=Pfin
FDAT_ACT=Fl064
BAS(#PTP_PARAMS,100)
PTP Xl064 C_DIS
;ENDFOLD
;FOLD PTP l066 CONT Vel=100 % fin Tool[5]:GUN C3 Base[3]:Atego/Axor;%{PE}%R 8.2.20,%MKUKATPBASIS,%CMOVE,%VPTP,%P 1:PTP, 2:l066, 3:C_DIS, 5:100, 7:fin
$BWDSTART=FALSE
PDAT_ACT=Pfin
FDAT_ACT=Fl066
BAS(#PTP_PARAMS,100)
PTP Xl066 C_DIS
;ENDFOLD

;FOLD ; SWP_60_9173;%{PE}%R 8.2.20,%MKUKATPBASIS,%CCOMMENT,%VNORMAL,%P 2:SWP_60_9173
;ENDFOLD
;FOLD PTP SWP_60_9173 vmax SPOT Gun=3 RETR CLS PgNo1=201 ACTIVE=1 Tool[5]:GUN C3 Base[3]:Atego/Axor;%{PE}%R 8.2.2,%MKUKATPSPOT,%CSPOT,%VPTP,%P 1:PTP, 2:SWP_60_9173, 3:, 5:100, 7:vmax, 10:3, 12:#FIRST, 14:#CLO, 16:201, 18:1, 20:0, 22:0, 24:1, 25:NORMAL
$BWDSTART=FALSE
PDAT_ACT=Pvmax
FDAT_ACT=FSWP_60_9173
BAS(#PTP_PARAMS,Pvmax.VEL)
S_ACT.GUN=3
S_ACT.PAIR=SDEFAULT.PAIR
S_ACT.RETR=#CLO
S_ACT.CLO_TM=1
S_ACT.PGNO1=201
S_ACT.PGNO2=SDEFAULT.PGNO2
S_ACT.PRESS1=SDEFAULT.PRESS1
S_ACT.PRESS2=SDEFAULT.PRESS2
S_READY=FALSE
PTP XSWP_60_9173
USERSPOT(#SPOT, S_ACT)
WAIT FOR S_READY
;ENDFOLD

;FOLD PTP P1 Vel=100 % fin Tool[5]:GUN C3 Base[3]:Atego/Axor;%{PE}%R 8.2.20,%MKUKATPBASIS,%CMOVE,%VPTP,%P 1:PTP, 2:P1, 3:, 5:100, 7:fin
$BWDSTART=FALSE
PDAT_ACT=Pfin
FDAT_ACT=FP1
BAS(#PTP_PARAMS,100)
PTP XP1
;ENDFOLD
;FOLD PTP P2 Vel=100 % fin Tool[5]:GUN C3 Base[3]:Atego/Axor;%{PE}%R 8.2.20,%MKUKATPBASIS,%CMOVE,%VPTP,%P 1:PTP, 2:P2, 3:, 5:100, 7:fin
$BWDSTART=FALSE
PDAT_ACT=Pfin
FDAT_ACT=FP2
BAS(#PTP_PARAMS,100)
PTP XP2
;ENDFOLD

;FOLD ; SWP_60_9175;%{PE}%R 8.2.20,%MKUKATPBASIS,%CCOMMENT,%VNORMAL,%P 2:SWP_60_9175
;ENDFOLD
;FOLD PTP SWP_60_9175 vmax SPOT Gun=3 RETR CLS PgNo1=201 ACTIVE=1 Tool[5]:GUN C3 Base[3]:Atego/Axor;%{PE}%R 8.2.2,%MKUKATPSPOT,%CSPOT,%VPTP,%P 1:PTP, 2:SWP_60_9175, 3:, 5:100, 7:vmax, 10:3, 12:#FIRST, 14:#CLO, 16:201, 18:1, 20:0, 22:0, 24:1, 25:NORMAL
$BWDSTART=FALSE
PDAT_ACT=Pvmax
FDAT_ACT=FSWP_60_9175
BAS(#PTP_PARAMS,Pvmax.VEL)
S_ACT.GUN=3
S_ACT.PAIR=SDEFAULT.PAIR
S_ACT.RETR=#CLO
S_ACT.CLO_TM=1
S_ACT.PGNO1=201
S_ACT.PGNO2=SDEFAULT.PGNO2
S_ACT.PRESS1=SDEFAULT.PRESS1
S_ACT.PRESS2=SDEFAULT.PRESS2
S_READY=FALSE
PTP XSWP_60_9175
USERSPOT(#SPOT, S_ACT)
WAIT FOR S_READY
;ENDFOLD

;FOLD ; SWP_60_9177;%{PE}%R 8.2.20,%MKUKATPBASIS,%CCOMMENT,%VNORMAL,%P 2:SWP_60_9177
;ENDFOLD
;FOLD PTP SWP_60_9177 vmax SPOT Gun=3 RETR CLS PgNo1=201 ACTIVE=1 Tool[5]:GUN C3 Base[3]:Atego/Axor;%{PE}%R 8.2.2,%MKUKATPSPOT,%CSPOT,%VPTP,%P 1:PTP, 2:SWP_60_9177, 3:, 5:100, 7:vmax, 10:3, 12:#FIRST, 14:#CLO, 16:201, 18:1, 20:0, 22:0, 24:1, 25:NORMAL
$BWDSTART=FALSE
PDAT_ACT=Pvmax
FDAT_ACT=FSWP_60_9177
BAS(#PTP_PARAMS,Pvmax.VEL)
S_ACT.GUN=3
S_ACT.PAIR=SDEFAULT.PAIR
S_ACT.RETR=#CLO
S_ACT.CLO_TM=1
S_ACT.PGNO1=201
S_ACT.PGNO2=SDEFAULT.PGNO2
S_ACT.PRESS1=SDEFAULT.PRESS1
S_ACT.PRESS2=SDEFAULT.PRESS2
S_READY=FALSE
PTP XSWP_60_9177
USERSPOT(#SPOT, S_ACT)
WAIT FOR S_READY
;ENDFOLD

;FOLD PTP l067 CONT Vel=100 % fin Tool[5]:GUN C3 Base[3]:Atego/Axor;%{PE}%R 8.2.20,%MKUKATPBASIS,%CMOVE,%VPTP,%P 1:PTP, 2:l067, 3:C_DIS, 5:100, 7:fin
$BWDSTART=FALSE
PDAT_ACT=Pfin
FDAT_ACT=Fl067
BAS(#PTP_PARAMS,100)
PTP Xl067 C_DIS
;ENDFOLD

;FOLD ; SWP_60_9181;%{PE}%R 8.2.20,%MKUKATPBASIS,%CCOMMENT,%VNORMAL,%P 2:SWP_60_9181
;ENDFOLD
;FOLD PTP SWP_60_9181 vmax SPOT Gun=3 RETR CLS PgNo1=201 ACTIVE=1 Tool[5]:GUN C3 Base[3]:Atego/Axor;%{PE}%R 8.2.2,%MKUKATPSPOT,%CSPOT,%VPTP,%P 1:PTP, 2:SWP_60_9181, 3:, 5:100, 7:vmax, 10:3, 12:#FIRST, 14:#CLO, 16:201, 18:1, 20:0, 22:0, 24:1, 25:NORMAL
$BWDSTART=FALSE
PDAT_ACT=Pvmax
FDAT_ACT=FSWP_60_9181
BAS(#PTP_PARAMS,Pvmax.VEL)
S_ACT.GUN=3
S_ACT.PAIR=SDEFAULT.PAIR
S_ACT.RETR=#CLO
S_ACT.CLO_TM=1
S_ACT.PGNO1=201
S_ACT.PGNO2=SDEFAULT.PGNO2
S_ACT.PRESS1=SDEFAULT.PRESS1
S_ACT.PRESS2=SDEFAULT.PRESS2
S_READY=FALSE
PTP XSWP_60_9181
USERSPOT(#SPOT, S_ACT)
WAIT FOR S_READY
;ENDFOLD

;FOLD ; SWP_60_9183;%{PE}%R 8.2.20,%MKUKATPBASIS,%CCOMMENT,%VNORMAL,%P 2:SWP_60_9183
;ENDFOLD
;FOLD PTP SWP_60_9183 vmax SPOT Gun=3 RETR CLS PgNo1=201 ACTIVE=1 Tool[5]:GUN C3 Base[3]:Atego/Axor;%{PE}%R 8.2.2,%MKUKATPSPOT,%CSPOT,%VPTP,%P 1:PTP, 2:SWP_60_9183, 3:, 5:100, 7:vmax, 10:3, 12:#FIRST, 14:#CLO, 16:201, 18:1, 20:0, 22:0, 24:1, 25:NORMAL
$BWDSTART=FALSE
PDAT_ACT=Pvmax
FDAT_ACT=FSWP_60_9183
BAS(#PTP_PARAMS,Pvmax.VEL)
S_ACT.GUN=3
S_ACT.PAIR=SDEFAULT.PAIR
S_ACT.RETR=#CLO
S_ACT.CLO_TM=1
S_ACT.PGNO1=201
S_ACT.PGNO2=SDEFAULT.PGNO2
S_ACT.PRESS1=SDEFAULT.PRESS1
S_ACT.PRESS2=SDEFAULT.PRESS2
S_READY=FALSE
PTP XSWP_60_9183
USERSPOT(#SPOT, S_ACT)
WAIT FOR S_READY
;ENDFOLD

;FOLD PTP P3 CONT Vel=100 % fin Tool[5]:GUN C3 Base[3]:Atego/Axor;%{PE}%R 8.2.20,%MKUKATPBASIS,%CMOVE,%VPTP,%P 1:PTP, 2:P3, 3:C_DIS, 5:100, 7:fin
$BWDSTART=FALSE
PDAT_ACT=Pfin
FDAT_ACT=FP3
BAS(#PTP_PARAMS,100)
PTP XP3 C_DIS
;ENDFOLD
;FOLD PTP P4 CONT Vel=100 % fin Tool[5]:GUN C3 Base[3]:Atego/Axor;%{PE}%R 8.2.20,%MKUKATPBASIS,%CMOVE,%VPTP,%P 1:PTP, 2:P4, 3:C_DIS, 5:100, 7:fin
$BWDSTART=FALSE
PDAT_ACT=Pfin
FDAT_ACT=FP4
BAS(#PTP_PARAMS,100)
PTP XP4 C_DIS
;ENDFOLD

;FOLD ; SWP_60_9185;%{PE}%R 8.2.20,%MKUKATPBASIS,%CCOMMENT,%VNORMAL,%P 2:SWP_60_9185
;ENDFOLD
;FOLD PTP SWP_60_9185 vmax SPOT Gun=3 RETR CLS PgNo1=201 ACTIVE=1 Tool[5]:GUN C3 Base[3]:Atego/Axor;%{PE}%R 8.2.2,%MKUKATPSPOT,%CSPOT,%VPTP,%P 1:PTP, 2:SWP_60_9185, 3:, 5:100, 7:vmax, 10:3, 12:#FIRST, 14:#CLO, 16:201, 18:1, 20:0, 22:0, 24:1, 25:NORMAL
$BWDSTART=FALSE
PDAT_ACT=Pvmax
FDAT_ACT=FSWP_60_9185
BAS(#PTP_PARAMS,Pvmax.VEL)
S_ACT.GUN=3
S_ACT.PAIR=SDEFAULT.PAIR
S_ACT.RETR=#CLO
S_ACT.CLO_TM=1
S_ACT.PGNO1=201
S_ACT.PGNO2=SDEFAULT.PGNO2
S_ACT.PRESS1=SDEFAULT.PRESS1
S_ACT.PRESS2=SDEFAULT.PRESS2
S_READY=FALSE
PTP XSWP_60_9185
USERSPOT(#SPOT, S_ACT)
WAIT FOR S_READY
;ENDFOLD

;FOLD ; Fim dos Pontos adicionados;%{PE}%R 8.2.20,%MKUKATPBASIS,%CCOMMENT,%VNORMAL,%P 2:Fim  dos  Pontos adicionados
;ENDFOLD

;FOLD PTP P7 CONT Vel=100 % fin Tool[5]:GUN C3 Base[3]:Atego/Axor;%{PE}%R 8.2.20,%MKUKATPBASIS,%CMOVE,%VPTP,%P 1:PTP, 2:P7, 3:C_DIS, 5:100, 7:fin
$BWDSTART=FALSE
PDAT_ACT=Pfin
FDAT_ACT=FP7
BAS(#PTP_PARAMS,100)
PTP XP7 C_DIS
;ENDFOLD
;FOLD PTP l068 CONT Vel=100 % small Tool[5]:GUN C3 Base[3]:Atego/Axor;%{PE}%R 8.2.20,%MKUKATPBASIS,%CMOVE,%VPTP,%P 1:PTP, 2:l068, 3:C_DIS, 5:100, 7:small
$BWDSTART=FALSE
PDAT_ACT=Psmall
FDAT_ACT=Fl068
BAS(#PTP_PARAMS,100)
PTP Xl068 C_DIS
;ENDFOLD
;FOLD PTP l069 CONT Vel=100 % xlarge Tool[5]:GUN C3 Base[3]:Atego/Axor;%{PE}%R 8.2.20,%MKUKATPBASIS,%CMOVE,%VPTP,%P 1:PTP, 2:l069, 3:C_DIS, 5:100, 7:xlarge
$BWDSTART=FALSE
PDAT_ACT=Pxlarge
FDAT_ACT=Fl069
BAS(#PTP_PARAMS,100)
PTP Xl069 C_DIS
;ENDFOLD
;FOLD PTP l035 CONT Vel=100 % xlarge Tool[5]:GUN C3 Base[3]:Atego/Axor;%{PE}%R 8.2.20,%MKUKATPBASIS,%CMOVE,%VPTP,%P 1:PTP, 2:l035, 3:C_DIS, 5:100, 7:xlarge
$BWDSTART=FALSE
PDAT_ACT=Pxlarge
FDAT_ACT=Fl035
BAS(#PTP_PARAMS,100)
PTP Xl035 C_DIS
;ENDFOLD
;FOLD PTP l013 Vel=100 % P_OLP38 Tool[5]:GUN C3 Base[3]:Atego/Axor;%{PE}%R 8.2.20,%MKUKATPBASIS,%CMOVE,%VPTP,%P 1:PTP, 2:l013, 3:, 5:100, 7:P_OLP38
$BWDSTART=FALSE
PDAT_ACT=PP_OLP38
FDAT_ACT=Fl013
BAS(#PTP_PARAMS,100)
PTP Xl013
;ENDFOLD


; FIM DE TRABALHO RESPOT
;FOLD PULSE 3333 'R3 trabalho concluído' State=TRUE Time=2 sec;%{PE}%R 8.2.20,%MKUKATPBASIS,%COUT,%VPULSE,%P 2:3333, 3:R3 trabalho concluído, 5:TRUE, 6:, 8:2
PULSE($OUT[3333], TRUE,2)
;ENDFOLD
;FOLD OUT 3348 'Fora area GEOBOX' State=TRUE ;%{PE}%R 8.2.20,%MKUKATPBASIS,%COUT,%VOUTX,%P 2:3348, 3:Fora area GEOBOX, 5:TRUE, 6:
$OUT[3348]=TRUE
;ENDFOLD

;FOLD SYN OUT 3340 'Area_clear_AGV' State=TRUE at START Delay=0 ms;%{PE}%R 8.2.20,%MKUKATPBASIS,%COUT,%VSYNOUT,%P 2:3340, 3:Area_clear_AGV, 5:TRUE, 7:0, 9:0, 12:0
TRIGGER WHEN DISTANCE=0 DELAY=0 DO $OUT[3340]=TRUE
;ENDFOLD
;FOLD ; DESLIGA INTERTRAVAMENTO 4 DE SEGURANCAO COM R4 COM A GARRA;%{PE}%R 8.2.20,%MKUKATPBASIS,%CCOMMENT,%VNORMAL,%P 2:DESLIGA  INTERTRAVAMENTO  4  DE  SEGURANCAO COM  R4  COM  A  GARRA
;ENDFOLD
;FOLD Collision.Monitoring_4_Off . ;%{PE}%MKUKATPUSER
COLLSTOP( 4, 2+0 )
;ENDFOLD

IF (NOT(GHOST())) THEN
if FraesAnf (3) then
f_fraes5 ()
endif
ENDIF

END

--- ps_b_etb_res_c03_R.dat ---
&ACCESS RVO2
&COMMENT Solda Atego STB
&PARAM DISKPATH = KRC:\R1\Program\olp
DEFDAT ps_b_etb_res_c03_R
;FOLD EXTERNAL DECLARATIONS;%{PE}%MKUKATPBASIS,%CEXT,%VCOMMON,%P
;FOLD GRIPPERTECH EXT
EXT  H50 (INT  :IN,INT  :IN,INT  :IN,GRP_TYP  :IN )
;ENDFOLD (GRIPPERTECH EXT)
;FOLD SPOTTECH EXT
EXT  USERSPOT (S_COMMAND  :IN,SPOT_TYPE  :IN )
;ENDFOLD (SPOTTECH EXT)
;FOLD BASISTECH EXT;%{PE}%MKUKATPBASIS,%CEXT,%VEXT,%P
EXT  BAS (BAS_COMMAND  :IN,REAL  :IN )
DECL INT SUCCESS
;ENDFOLD (BASISTECH EXT)
;FOLD USER EXT;%{E}%MKUKATPUSER,%CEXT,%VEXT,%P
;Make your modifications here

;ENDFOLD (USER EXT)
;ENDFOLD (EXTERNAL DECLARATIONS)
DECL FDAT Fl010={TOOL_NO 5,BASE_NO 3,IPO_FRAME #BASE,POINT2[] " "}
DECL PDAT PP_OLP3={VEL 100.0,ACC 100.0,APO_DIST 100.0,APO_MODE #CDIS}
DECL E6POS Xl010={X 192.420197,Y -166.267899,Z 148.271805,A 93.6815338,B -3.17932296,C -90.3057938,S 2,T 35,E1 4299.99023,E2 0.0,E3 0.0,E4 0.0,E5 0.0,E6 0.0}
DECL FDAT Fl035={TOOL_NO 5,BASE_NO 3,IPO_FRAME #BASE,POINT2[] " "}
DECL PDAT PP_OLP8={VEL 100.0,ACC 100.0,APO_DIST 100.0,APO_MODE #CDIS}
DECL E6POS Xl035={X -688.517822,Y -889.36792,Z -9.54666424,A -69.0801468,B -9.38054085,C 48.8003082,S 2,T 35,E1 4299.99707,E2 0.0,E3 0.0,E4 0.0,E5 0.0,E6 0.0}
DECL BASIS_SUGG_T LAST_BASIS={POINT1[] "P7                      ",POINT2[] "P7                      ",CP_PARAMS[] "CPDAT0                  ",PTP_PARAMS[] "PDAT6                   ",CONT[] "C_DIS                   ",CP_VEL[] "2.0                     ",PTP_VEL[] "100                     ",SYNC_PARAMS[] "SYNCDAT                 ",SPL_NAME[] "S0                      "}
DECL PDAT PP_OLP14={VEL 100.0,ACC 100.0,APO_DIST 100.0,APO_MODE #CDIS}
DECL E6POS Xl016={X -1200.354,Y -1467.33997,Z -420.136902,A 6.10609007,B -34.4457092,C -4.04726219,S 2,T 35,E1 3455.71802,E2 0.0,E3 0.0,E4 0.0,E5 0.0,E6 0.0}
DECL FDAT Fl016={TOOL_NO 5,BASE_NO 3,IPO_FRAME #BASE,POINT2[] " "}
DECL PDAT PP_OLP15={VEL 100.0,ACC 100.0,APO_DIST 10.0,APO_MODE #CDIS}
DECL E6POS Xl021={X -504.116486,Y -800.927429,Z -215.553894,A -24.5715904,B -53.4077797,C 26.2354107,S 2,T 35,E1 4300.0,E2 0.0,E3 0.0,E4 0.0,E5 0.0,E6 0.0}
DECL FDAT Fl021={TOOL_NO 5,BASE_NO 3,IPO_FRAME #BASE,POINT2[] " "}
DECL PDAT PP_OLP16={VEL 100.0,ACC 100.0,APO_DIST 10.0,APO_MODE #CDIS}
DECL E6POS Xl026={X 105.730904,Y -605.006104,Z -121.837402,A -88.0092926,B -76.6820602,C 92.2949066,S 2,T 35,E1 4299.99902,E2 0.0,E3 0.0,E4 0.0,E5 0.0,E6 0.0}
DECL FDAT Fl026={TOOL_NO 5,BASE_NO 3,IPO_FRAME #BASE,POINT2[] " "}
DECL PDAT PP_OLP17={VEL 100.0,ACC 100.0,APO_DIST 10.0,APO_MODE #CDIS}
DECL E6POS Xl031={X 197.095596,Y -842.804382,Z -195.312195,A -87.0241623,B -80.1558533,C 88.4448624,S 2,T 35,E1 4300.00195,E2 0.0,E3 0.0,E4 0.0,E5 0.0,E6 0.0}
DECL FDAT Fl031={TOOL_NO 5,BASE_NO 3,IPO_FRAME #BASE,POINT2[] " "}
DECL LDAT LL_OLP3={VEL 2.0,ACC 100.0,APO_DIST 0.0,APO_FAC 0.0,ORI_TYP #VAR,CIRC_TYP #BASE,JERK_FAC 50.0}
DECL E6POS XSWP_60_7053={X 192.730392,Y -882.800476,Z -187.645203,A -89.9909134,B -79.9946594,C 89.9927597,S 2,T 35,E1 4300.00195,E2 0.0,E3 0.0,E4 0.0,E5 0.0,E6 0.0}
DECL FDAT FSWP_60_7053={TOOL_NO 5,BASE_NO 3,IPO_FRAME #BASE,POINT2[] " "}
DECL PDAT PP_OLP19={VEL 100.0,ACC 100.0,APO_DIST 100.0,APO_MODE #CDIS}
DECL E6POS Xl041={X 197.749405,Y -857.262024,Z -180.264008,A -89.9999924,B -80.0000992,C 89.9999924,S 2,T 35,E1 4300.0,E2 0.0,E3 0.0,E4 0.0,E5 0.0,E6 0.0}
DECL FDAT Fl041={TOOL_NO 5,BASE_NO 3,IPO_FRAME #BASE,POINT2[] " "}
DECL LDAT LL_OLP4={VEL 2.0,ACC 100.0,APO_DIST 0.0,APO_FAC 0.0,ORI_TYP #VAR,CIRC_TYP #BASE,JERK_FAC 50.0}
DECL E6POS XSWP_60_7051={X 192.190796,Y -853.006714,Z -159.147797,A -89.9849777,B -79.9993362,C 89.9846191,S 2,T 35,E1 4300.00781,E2 0.0,E3 0.0,E4 0.0,E5 0.0,E6 0.0}
DECL FDAT FSWP_60_7051={TOOL_NO 5,BASE_NO 3,IPO_FRAME #BASE,POINT2[] " "}
DECL LDAT LL_OLP5={VEL 2.0,ACC 100.0,APO_DIST 0.0,APO_FAC 0.0,ORI_TYP #VAR,CIRC_TYP #BASE,JERK_FAC 50.0}
DECL E6POS XSWP_60_7049={X 192.047394,Y -824.388977,Z -130.335602,A -90.0232315,B -79.9922714,C 90.0233917,S 2,T 35,E1 4300.00781,E2 0.0,E3 0.0,E4 0.0,E5 0.0,E6 0.0}
DECL FDAT FSWP_60_7049={TOOL_NO 5,BASE_NO 3,IPO_FRAME #BASE,POINT2[] " "}
DECL LDAT LL_OLP6={VEL 2.0,ACC 100.0,APO_DIST 0.0,APO_FAC 0.0,ORI_TYP #VAR,CIRC_TYP #BASE,JERK_FAC 50.0}
DECL E6POS XSWP_60_7047={X 192.727097,Y -795.518616,Z -101.527298,A -90.0249176,B -79.9941635,C 90.024353,S 2,T 35,E1 4299.979,E2 0.0,E3 0.0,E4 0.0,E5 0.0,E6 0.0}
DECL FDAT FSWP_60_7047={TOOL_NO 5,BASE_NO 3,IPO_FRAME #BASE,POINT2[] " "}
DECL LDAT LL_OLP7={VEL 2.0,ACC 100.0,APO_DIST 0.0,APO_FAC 0.0,ORI_TYP #VAR,CIRC_TYP #BASE,JERK_FAC 50.0}
DECL E6POS XSWP_60_7045={X 190.991699,Y -769.520874,Z -74.9092331,A -90.0168304,B -80.0018311,C 90.0171814,S 2,T 35,E1 4299.98682,E2 0.0,E3 0.0,E4 0.0,E5 0.0,E6 0.0}
DECL FDAT FSWP_60_7045={TOOL_NO 5,BASE_NO 3,IPO_FRAME #BASE,POINT2[] " "}
DECL PDAT PP_OLP20={VEL 100.0,ACC 100.0,APO_DIST 100.0,APO_MODE #CDIS}
DECL E6POS Xl046={X 201.858704,Y -724.052979,Z -74.0759964,A 89.9998016,B -85.0,C -90.0,S 2,T 35,E1 4300.0,E2 0.0,E3 0.0,E4 0.0,E5 0.0,E6 0.0}
DECL FDAT Fl046={TOOL_NO 5,BASE_NO 3,IPO_FRAME #BASE,POINT2[] " "}
DECL LDAT LL_OLP8={VEL 2.0,ACC 100.0,APO_DIST 0.0,APO_FAC 0.0,ORI_TYP #VAR,CIRC_TYP #BASE,JERK_FAC 50.0}
DECL E6POS XSWP_60_7041={X 191.9142,Y -697.815674,Z -49.9122505,A 90.0055695,B -65.0068436,C -89.9991074,S 2,T 35,E1 4300.03076,E2 0.0,E3 0.0,E4 0.0,E5 0.0,E6 0.0}
DECL FDAT FSWP_60_7041={TOOL_NO 5,BASE_NO 3,IPO_FRAME #BASE,POINT2[] " "}
DECL LDAT LL_OLP9={VEL 2.0,ACC 100.0,APO_DIST 0.0,APO_FAC 0.0,ORI_TYP #VAR,CIRC_TYP #BASE,JERK_FAC 50.0}
DECL E6POS XSWP_60_7039={X 190.732803,Y -659.745789,Z -55.9621696,A 89.9975815,B -65.006691,C -89.9963226,S 2,T 35,E1 4300.00293,E2 0.0,E3 0.0,E4 0.0,E5 0.0,E6 0.0}
DECL FDAT FSWP_60_7039={TOOL_NO 5,BASE_NO 3,IPO_FRAME #BASE,POINT2[] " "}
DECL LDAT LL_OLP10={VEL 2.0,ACC 100.0,APO_DIST 0.0,APO_FAC 0.0,ORI_TYP #VAR,CIRC_TYP #BASE,JERK_FAC 50.0}
DECL E6POS XSWP_60_7037={X 190.393997,Y -623.188171,Z -72.8631592,A 90.0108032,B -65.0110321,C -90.0050583,S 2,T 35,E1 4299.9541,E2 0.0,E3 0.0,E4 0.0,E5 0.0,E6 0.0}
DECL FDAT FSWP_60_7037={TOOL_NO 5,BASE_NO 3,IPO_FRAME #BASE,POINT2[] " "}
DECL LDAT LL_OLP11={VEL 2.0,ACC 100.0,APO_DIST 0.0,APO_FAC 0.0,ORI_TYP #VAR,CIRC_TYP #BASE,JERK_FAC 50.0}
DECL E6POS XSWP_60_7035={X 193.7789,Y -600.831482,Z -92.8529663,A 90.0178909,B -65.0057373,C -90.0168228,S 2,T 35,E1 4300.01611,E2 0.0,E3 0.0,E4 0.0,E5 0.0,E6 0.0}
DECL FDAT FSWP_60_7035={TOOL_NO 5,BASE_NO 3,IPO_FRAME #BASE,POINT2[] " "}
DECL PDAT PP_OLP22={VEL 100.0,ACC 100.0,APO_DIST 100.0,APO_MODE #CDIS}
DECL E6POS Xl055={X 189.028702,Y -635.804077,Z -124.194099,A 87.8480377,B -65.227211,C -87.4349365,S 2,T 35,E1 4300.01611,E2 0.0,E3 0.0,E4 0.0,E5 0.0,E6 0.0}
DECL FDAT Fl055={TOOL_NO 5,BASE_NO 3,IPO_FRAME #BASE,POINT2[] " "}
DECL PDAT PP_OLP23={VEL 100.0,ACC 100.0,APO_DIST 100.0,APO_MODE #CDIS}
DECL E6POS Xl060={X 74.9870682,Y -601.914429,Z -132.6017,A -86.6061935,B -78.2498398,C 90.0065765,S 2,T 35,E1 4300.0,E2 0.0,E3 0.0,E4 0.0,E5 0.0,E6 0.0}
DECL FDAT Fl060={TOOL_NO 5,BASE_NO 3,IPO_FRAME #BASE,POINT2[] " "}
DECL PDAT PP_OLP24={VEL 100.0,ACC 100.0,APO_DIST 100.0,APO_MODE #CDIS}
DECL E6POS Xl065={X 73.9980011,Y -296.309692,Z 79.4658813,A -90.0,B -25.0,C 90.0,S 2,T 35,E1 4300.0,E2 0.0,E3 0.0,E4 0.0,E5 0.0,E6 0.0}
DECL FDAT Fl065={TOOL_NO 5,BASE_NO 3,IPO_FRAME #BASE,POINT2[] " "}
DECL PDAT PP_OLP25={VEL 100.0,ACC 100.0,APO_DIST 100.0,APO_MODE #CDIS}
DECL E6POS Xl070={X 182.498993,Y -305.85199,Z 59.0,A -90.0,B 0.0,C 90.0,S 2,T 35,E1 4300.0,E2 0.0,E3 0.0,E4 0.0,E5 0.0,E6 0.0}
DECL FDAT Fl070={TOOL_NO 5,BASE_NO 3,IPO_FRAME #BASE,POINT2[] " "}
DECL PDAT PP_OLP26={VEL 100.0,ACC 100.0,APO_DIST 100.0,APO_MODE #CDIS}
DECL E6POS Xl075={X 179.639297,Y -350.85199,Z 58.9990005,A -90.0,B -1.36636604E-08,C 90.0,S 2,T 35,E1 4300.0,E2 0.0,E3 0.0,E4 0.0,E5 0.0,E6 0.0}
DECL FDAT Fl075={TOOL_NO 5,BASE_NO 3,IPO_FRAME #BASE,POINT2[] " "}
DECL PDAT PP_OLP27={VEL 100.0,ACC 100.0,APO_DIST 100.0,APO_MODE #CDIS}
DECL E6POS Xl080={X 177.080307,Y -320.852997,Z 73.9970016,A -90.0,B -3.01534087E-08,C 90.0,S 2,T 35,E1 4300.0,E2 0.0,E3 0.0,E4 0.0,E5 0.0,E6 0.0}
DECL FDAT Fl080={TOOL_NO 5,BASE_NO 3,IPO_FRAME #BASE,POINT2[] " "}
DECL PDAT PP_OLP28={VEL 100.0,ACC 100.0,APO_DIST 100.0,APO_MODE #CDIS}
DECL E6POS Xl085={X 174.526398,Y -312.003998,Z 147.546005,A -90.0,B -5.00010014,C 90.0,S 2,T 35,E1 4300.0,E2 0.0,E3 0.0,E4 0.0,E5 0.0,E6 0.0}
DECL FDAT Fl085={TOOL_NO 5,BASE_NO 3,IPO_FRAME #BASE,POINT2[] " "}
DECL LDAT LL_OLP13={VEL 2.0,ACC 100.0,APO_DIST 0.0,APO_FAC 0.0,ORI_TYP #VAR,CIRC_TYP #BASE,JERK_FAC 50.0}
DECL E6POS XSWP_60_7127={X 176.629303,Y -353.700104,Z 159.217102,A -91.2654037,B -4.81602192,C 90.1614304,S 2,T 35,E1 4300.00586,E2 0.0,E3 0.0,E4 0.0,E5 0.0,E6 0.0}
DECL FDAT FSWP_60_7127={TOOL_NO 5,BASE_NO 3,IPO_FRAME #BASE,POINT2[] " "}
DECL LDAT LL_OLP15={VEL 2.0,ACC 100.0,APO_DIST 0.0,APO_FAC 0.0,ORI_TYP #VAR,CIRC_TYP #BASE,JERK_FAC 50.0}
DECL E6POS XSWP_60_7129={X 175.556702,Y -351.091187,Z 187.268204,A -90.0573883,B -5.00000095,C 89.454071,S 2,T 35,E1 4300.0,E2 0.0,E3 0.0,E4 0.0,E5 0.0,E6 0.0}
DECL FDAT FSWP_60_7129={TOOL_NO 5,BASE_NO 3,IPO_FRAME #BASE,POINT2[] " "}
DECL LDAT LL_OLP16={VEL 2.0,ACC 100.0,APO_DIST 0.0,APO_FAC 0.0,ORI_TYP #VAR,CIRC_TYP #BASE,JERK_FAC 50.0}
DECL E6POS XSWP_60_7131={X 175.778397,Y -346.909698,Z 217.144806,A -90.031723,B -10.2092695,C 89.7102737,S 2,T 35,E1 4299.96924,E2 0.0,E3 0.0,E4 0.0,E5 0.0,E6 0.0}
DECL FDAT FSWP_60_7131={TOOL_NO 5,BASE_NO 3,IPO_FRAME #BASE,POINT2[] " "}
DECL LDAT LL_OLP17={VEL 2.0,ACC 100.0,APO_DIST 0.0,APO_FAC 0.0,ORI_TYP #VAR,CIRC_TYP #BASE,JERK_FAC 50.0}
DECL E6POS XSWP_60_7133={X 176.018906,Y -336.620789,Z 244.570297,A -90.0156174,B -10.1044903,C 89.8553314,S 2,T 35,E1 4299.97803,E2 0.0,E3 0.0,E4 0.0,E5 0.0,E6 0.0}
DECL FDAT FSWP_60_7133={TOOL_NO 5,BASE_NO 3,IPO_FRAME #BASE,POINT2[] " "}
DECL LDAT LL_OLP18={VEL 2.0,ACC 100.0,APO_DIST 0.0,APO_FAC 0.0,ORI_TYP #VAR,CIRC_TYP #BASE,JERK_FAC 50.0}
DECL E6POS XSWP_60_7135={X 176.0811,Y -321.196899,Z 266.562408,A -90.0093536,B -17.1961708,C 89.9071198,S 2,T 35,E1 4299.98584,E2 0.0,E3 0.0,E4 0.0,E5 0.0,E6 0.0}
DECL FDAT FSWP_60_7135={TOOL_NO 5,BASE_NO 3,IPO_FRAME #BASE,POINT2[] " "}
DECL LDAT LL_OLP19={VEL 2.0,ACC 100.0,APO_DIST 0.0,APO_FAC 0.0,ORI_TYP #VAR,CIRC_TYP #BASE,JERK_FAC 50.0}
DECL E6POS XSWP_60_7139={X 175.219498,Y -276.463287,Z 293.379211,A -90.002861,B -26.2956104,C 89.9732971,S 2,T 35,E1 4299.99609,E2 0.0,E3 0.0,E4 0.0,E5 0.0,E6 0.0}
DECL FDAT FSWP_60_7139={TOOL_NO 5,BASE_NO 3,IPO_FRAME #BASE,POINT2[] " "}
DECL LDAT LL_OLP20={VEL 2.0,ACC 100.0,APO_DIST 0.0,APO_FAC 0.0,ORI_TYP #VAR,CIRC_TYP #BASE,JERK_FAC 50.0}
DECL E6POS XSWP_60_7143={X 176.370499,Y -237.512695,Z 295.863403,A -90.0068665,B -45.0004807,C 90.0071487,S 2,T 35,E1 4300.0,E2 0.0,E3 0.0,E4 0.0,E5 0.0,E6 0.0}
DECL FDAT FSWP_60_7143={TOOL_NO 5,BASE_NO 3,IPO_FRAME #BASE,POINT2[] " "}
DECL LDAT LL_OLP21={VEL 2.0,ACC 100.0,APO_DIST 0.0,APO_FAC 0.0,ORI_TYP #VAR,CIRC_TYP #BASE,JERK_FAC 50.0}
DECL E6POS XSWP_60_7153={X 175.899399,Y -69.6962128,Z 299.700897,A -89.9997177,B -30.0000591,C 89.9988174,S 2,T 35,E1 4300.0,E2 0.0,E3 0.0,E4 0.0,E5 0.0,E6 0.0}
DECL FDAT FSWP_60_7153={TOOL_NO 5,BASE_NO 3,IPO_FRAME #BASE,POINT2[] " "}
DECL LDAT LL_OLP22={VEL 2.0,ACC 100.0,APO_DIST 0.0,APO_FAC 0.0,ORI_TYP #VAR,CIRC_TYP #BASE,JERK_FAC 50.0}
DECL E6POS XSWP_60_7155={X 176.539993,Y -36.9459991,Z 300.688385,A -90.0000229,B -29.9999504,C 89.9999313,S 2,T 35,E1 4300.0,E2 0.0,E3 0.0,E4 0.0,E5 0.0,E6 0.0}
DECL FDAT FSWP_60_7155={TOOL_NO 5,BASE_NO 3,IPO_FRAME #BASE,POINT2[] " "}
DECL LDAT LL_OLP23={VEL 2.0,ACC 100.0,APO_DIST 0.0,APO_FAC 0.0,ORI_TYP #VAR,CIRC_TYP #BASE,JERK_FAC 50.0}
DECL E6POS XSWP_60_7157={X 174.774307,Y -2.6844039,Z 300.079987,A -90.0000229,B -29.9999504,C 89.9999313,S 2,T 35,E1 4300.0,E2 0.0,E3 0.0,E4 0.0,E5 0.0,E6 0.0}
DECL FDAT FSWP_60_7157={TOOL_NO 5,BASE_NO 3,IPO_FRAME #BASE,POINT2[] " "}
DECL PDAT PP_OLP34={VEL 100.0,ACC 100.0,APO_DIST 100.0,APO_MODE #CDIS}
DECL E6POS Xl115={X 174.771805,Y -125.414497,Z 231.551697,A -89.9999771,B -29.9999504,C 89.9999084,S 2,T 35,E1 4300.0,E2 0.0,E3 0.0,E4 0.0,E5 0.0,E6 0.0}
DECL FDAT Fl115={TOOL_NO 5,BASE_NO 3,IPO_FRAME #BASE,POINT2[] " "}
DECL SPOT_SUGG_T LAST_SPOT={GUN[] "1                       ",RETR_CMD[] "#OPN                    ",CHOISE[] "#FIRST                  ",CLO_TM[] "0                       ",PGNO1[] "1                       ",PRESS1[] "0                       ",PGNO2[] "1                       ",PRESS2[] "0                       ",SPOT_PARAMS[] "NORMAL                  "}
DECL PDAT PP_OLP37={VEL 100.0,ACC 100.0,APO_DIST 10.0,APO_MODE #CDIS}
DECL E6POS Xl012={X -1945.76794,Y -1816.99695,Z -419.417786,A -0.634959877,B 0.0284670591,C 0.673866689,S 2,T 43,E1 3416.84399,E2 0.0,E3 0.0,E4 0.0,E5 0.0,E6 0.0}
DECL FDAT Fl012={TOOL_NO 5,BASE_NO 3,IPO_FRAME #BASE,POINT2[] " "}
DECL PDAT PP_OLP38={VEL 100.0,ACC 100.0,APO_DIST 10.0,APO_MODE #CDIS}
DECL E6POS Xl013={X -1945.67896,Y -1816.92603,Z -419.428009,A -0.639662504,B 0.0256760698,C 0.675719976,S 2,T 43,E1 3416.85303,E2 0.0,E3 0.0,E4 0.0,E5 0.0,E6 0.0}
DECL FDAT Fl013={TOOL_NO 5,BASE_NO 3,IPO_FRAME #BASE,POINT2[] " "}
DECL LDAT LL_OLP26={VEL 2.0,ACC 100.0,APO_DIST 0.0,APO_FAC 0.0,ORI_TYP #VAR,CIRC_TYP #BASE,JERK_FAC 50.0}
DECL E6POS XSWP_60_7141={X 175.494293,Y -253.669403,Z 295.777802,A -89.9942932,B -41.5514984,C 89.9699478,S 2,T 35,E1 4299.99512,E2 0.0,E3 0.0,E4 0.0,E5 0.0,E6 0.0}
DECL FDAT FSWP_60_7141={TOOL_NO 5,BASE_NO 3,IPO_FRAME #BASE,POINT2[] " ",TQ_STATE FALSE}
DECL PDAT PP_OLP40={VEL 100.0,ACC 100.0,APO_DIST 100.0,APO_MODE #CDIS}
DECL E6POS Xl014={X 178.645493,Y -15.0816002,Z -17.3036308,A 89.2547379,B 84.585083,C -91.5456085,S 2,T 3,E1 4299.99219,E2 0.0,E3 0.0,E4 0.0,E5 0.0,E6 0.0}
DECL FDAT Fl014={TOOL_NO 5,BASE_NO 3,IPO_FRAME #BASE,POINT2[] " "}
DECL LDAT LL_OLP27={VEL 2.0,ACC 100.0,APO_DIST 0.0,APO_FAC 0.0,ORI_TYP #VAR,CIRC_TYP #BASE,JERK_FAC 50.0}
DECL LDAT LL_OLP28={VEL 2.0,ACC 100.0,APO_DIST 0.0,APO_FAC 0.0,ORI_TYP #VAR,CIRC_TYP #BASE,JERK_FAC 50.0}
DECL LDAT LL_OLP29={VEL 2.0,ACC 100.0,APO_DIST 0.0,APO_FAC 0.0,ORI_TYP #VAR,CIRC_TYP #BASE,JERK_FAC 50.0}
DECL E6POS XSWP_60_9150={X 169.6138,Y -103.885201,Z -46.4488602,A 89.2617035,B 84.5840683,C -91.5384827,S 2,T 3,E1 4299.98877,E2 0.0,E3 0.0,E4 0.0,E5 0.0,E6 0.0}
DECL FDAT FSWP_60_9150={TOOL_NO 5,BASE_NO 3,IPO_FRAME #BASE,POINT2[] " "}
DECL LDAT LL_OLP30={VEL 2.0,ACC 100.0,APO_DIST 0.0,APO_FAC 0.0,ORI_TYP #VAR,CIRC_TYP #BASE,JERK_FAC 50.0}
DECL LDAT LL_OLP31={VEL 2.0,ACC 100.0,APO_DIST 0.0,APO_FAC 0.0,ORI_TYP #VAR,CIRC_TYP #BASE,JERK_FAC 50.0}
DECL LDAT LL_OLP32={VEL 2.0,ACC 100.0,APO_DIST 0.0,APO_FAC 0.0,ORI_TYP #VAR,CIRC_TYP #BASE,JERK_FAC 50.0}
DECL LDAT LL_OLP33={VEL 2.0,ACC 100.0,APO_DIST 0.0,APO_FAC 0.0,ORI_TYP #VAR,CIRC_TYP #BASE,JERK_FAC 50.0}
DECL LDAT LL_OLP34={VEL 2.0,ACC 100.0,APO_DIST 0.0,APO_FAC 0.0,ORI_TYP #VAR,CIRC_TYP #BASE,JERK_FAC 50.0}
DECL LDAT LL_OLP35={VEL 2.0,ACC 100.0,APO_DIST 0.0,APO_FAC 0.0,ORI_TYP #VAR,CIRC_TYP #BASE,JERK_FAC 50.0}
DECL LDAT LL_OLP36={VEL 2.0,ACC 100.0,APO_DIST 0.0,APO_FAC 0.0,ORI_TYP #VAR,CIRC_TYP #BASE,JERK_FAC 50.0}
DECL PDAT PP_OLP41={VEL 100.0,ACC 100.0,APO_DIST 100.0,APO_MODE #CDIS}
DECL E6POS Xl032={X 168.900604,Y -271.340607,Z 76.1519394,A -89.0555725,B 46.2203903,C 90.2092438,S 2,T 3,E1 4299.98389,E2 0.0,E3 0.0,E4 0.0,E5 0.0,E6 0.0}
DECL FDAT Fl032={TOOL_NO 5,BASE_NO 3,IPO_FRAME #BASE,POINT2[] " "}
DECL PDAT PP_OLP42={VEL 100.0,ACC 100.0,APO_DIST 100.0,APO_MODE #CDIS}
DECL E6POS Xl033={X 14.1120396,Y -278.348694,Z 74.4917068,A -89.0556335,B 46.2204819,C 90.2092819,S 2,T 3,E1 4299.98291,E2 0.0,E3 0.0,E4 0.0,E5 0.0,E6 0.0}
DECL FDAT Fl033={TOOL_NO 5,BASE_NO 3,IPO_FRAME #BASE,POINT2[] " "}
DECL PDAT PP_OLP43={VEL 100.0,ACC 100.0,APO_DIST 100.0,APO_MODE #CDIS}
DECL E6POS Xl061={X 75.5903778,Y -664.025513,Z 135.634598,A -83.7556,B 3.29721999,C 90.8231277,S 2,T 35,E1 4300.00195,E2 0.0,E3 0.0,E4 0.0,E5 0.0,E6 0.0}
DECL FDAT Fl061={TOOL_NO 5,BASE_NO 3,IPO_FRAME #BASE,POINT2[] " "}
DECL PDAT PP_OLP44={VEL 100.0,ACC 100.0,APO_DIST 100.0,APO_MODE #CDIS}
DECL E6POS Xl062={X 201.605392,Y -797.531677,Z 135.590393,A -89.1518707,B 3.29826689,C 90.8205872,S 2,T 35,E1 4300.00195,E2 0.0,E3 0.0,E4 0.0,E5 0.0,E6 0.0}
DECL FDAT Fl062={TOOL_NO 5,BASE_NO 3,IPO_FRAME #BASE,POINT2[] " "}
DECL LDAT LL_OLP41={VEL 2.0,ACC 100.0,APO_DIST 0.0,APO_FAC 0.0,ORI_TYP #VAR,CIRC_TYP #BASE,JERK_FAC 50.0}
DECL LDAT LL_OLP42={VEL 2.0,ACC 100.0,APO_DIST 0.0,APO_FAC 0.0,ORI_TYP #VAR,CIRC_TYP #BASE,JERK_FAC 50.0}
DECL LDAT LL_OLP43={VEL 2.0,ACC 100.0,APO_DIST 0.0,APO_FAC 0.0,ORI_TYP #VAR,CIRC_TYP #BASE,JERK_FAC 50.0}
DECL LDAT LL_OLP44={VEL 2.0,ACC 100.0,APO_DIST 0.0,APO_FAC 0.0,ORI_TYP #VAR,CIRC_TYP #BASE,JERK_FAC 50.0}
DECL LDAT LL_OLP45={VEL 2.0,ACC 100.0,APO_DIST 0.0,APO_FAC 0.0,ORI_TYP #VAR,CIRC_TYP #BASE,JERK_FAC 50.0}
DECL LDAT LL_OLP46={VEL 2.0,ACC 100.0,APO_DIST 0.0,APO_FAC 0.0,ORI_TYP #VAR,CIRC_TYP #BASE,JERK_FAC 50.0}
DECL LDAT LL_OLP47={VEL 2.0,ACC 100.0,APO_DIST 0.0,APO_FAC 0.0,ORI_TYP #VAR,CIRC_TYP #BASE,JERK_FAC 50.0}
DECL PDAT PP_OLP46={VEL 100.0,ACC 100.0,APO_DIST 100.0,APO_MODE #CDIS}
DECL E6POS Xl064={X 209.228302,Y -816.362427,Z 104.588097,A -89.8272629,B 8.27282047,C 89.6189117,S 2,T 35,E1 4300.00195,E2 0.0,E3 0.0,E4 0.0,E5 0.0,E6 0.0}
DECL FDAT Fl064={TOOL_NO 5,BASE_NO 3,IPO_FRAME #BASE,POINT2[] " "}
DECL PDAT PP_OLP47={VEL 100.0,ACC 100.0,APO_DIST 100.0,APO_MODE #CDIS}
DECL E6POS Xl066={X 201.724106,Y -810.847778,Z 71.9489594,A -89.405098,B 25.8556194,C 90.5272903,S 2,T 35,E1 4299.98877,E2 0.0,E3 0.0,E4 0.0,E5 0.0,E6 0.0}
DECL FDAT Fl066={TOOL_NO 5,BASE_NO 3,IPO_FRAME #BASE,POINT2[] " "}
DECL PDAT PP_OLP48={VEL 100.0,ACC 100.0,APO_DIST 100.0,APO_MODE #CDIS}
DECL E6POS Xl067={X 207.444305,Y -685.201416,Z 33.6865387,A -90.0009766,B 80.518959,C 89.9987564,S 2,T 35,E1 4299.99805,E2 0.0,E3 0.0,E4 0.0,E5 0.0,E6 0.0}
DECL FDAT Fl067={TOOL_NO 5,BASE_NO 3,IPO_FRAME #BASE,POINT2[] " "}
DECL PDAT PP_OLP49={VEL 100.0,ACC 100.0,APO_DIST 100.0,APO_MODE #CDIS}
DECL E6POS Xl068={X 210.307693,Y -599.171021,Z 64.023613,A 89.9927673,B 55.4556808,C -90.0019836,S 2,T 35,E1 4299.99707,E2 0.0,E3 0.0,E4 0.0,E5 0.0,E6 0.0}
DECL FDAT Fl068={TOOL_NO 5,BASE_NO 3,IPO_FRAME #BASE,POINT2[] " "}
DECL PDAT PP_OLP50={VEL 100.0,ACC 100.0,APO_DIST 10.0,APO_MODE #CDIS}
DECL E6POS Xl069={X 23.9933796,Y -648.789612,Z 95.1425018,A -89.998909,B 57.9658813,C 89.9998322,S 2,T 35,E1 4299.99805,E2 0.0,E3 0.0,E4 0.0,E5 0.0,E6 0.0}
DECL FDAT Fl069={TOOL_NO 5,BASE_NO 3,IPO_FRAME #BASE,POINT2[] " "}
DECL PDAT PP_OLP51={VEL 100.0,ACC 100.0,APO_DIST 100.0,APO_MODE #CDIS}
DECL E6POS Xl034={X 16.2978001,Y -427.894592,Z 28.0205498,A 90.8066483,B -5.24551201,C -90.1453934,S 2,T 35,E1 4299.98291,E2 0.0,E3 0.0,E4 0.0,E5 0.0,E6 0.0}
DECL FDAT Fl034={TOOL_NO 5,BASE_NO 3,IPO_FRAME #BASE,POINT2[] " "}
DECL PDAT PP_OLP52={VEL 100.0,ACC 100.0,APO_DIST 10.0,APO_MODE #CDIS}
DECL E6POS Xl037={X 55.2557297,Y -277.908508,Z -176.818604,A -91.8772507,B -85.3020096,C 100.737503,S 2,T 35,E1 4299.98096,E2 0.0,E3 0.0,E4 0.0,E5 0.0,E6 0.0}
DECL FDAT Fl037={TOOL_NO 5,BASE_NO 3,IPO_FRAME #BASE,POINT2[] " "}
DECL PDAT PP_OLP53={VEL 100.0,ACC 100.0,APO_DIST 100.0,APO_MODE #CDIS}
DECL E6POS Xl038={X 184.757904,Y -268.897186,Z -158.233597,A -92.0511169,B -85.2995834,C 104.0205,S 2,T 35,E1 4299.979,E2 0.0,E3 0.0,E4 0.0,E5 0.0,E6 0.0}
DECL FDAT Fl038={TOOL_NO 5,BASE_NO 3,IPO_FRAME #BASE,POINT2[] " "}
DECL LDAT LL_OLP48={VEL 2.0,ACC 100.0,APO_DIST 0.0,APO_FAC 0.0,ORI_TYP #VAR,CIRC_TYP #BASE,JERK_FAC 50.0}
DECL PDAT PP_OLP54={VEL 100.0,ACC 100.0,APO_DIST 100.0,APO_MODE #CDIS}
DECL E6POS Xl039={X 184.757904,Y -268.897186,Z -158.233597,A -92.0511169,B -85.2995834,C 104.0205,S 2,T 35,E1 4299.979,E2 0.0,E3 0.0,E4 0.0,E5 0.0,E6 0.0}
DECL FDAT Fl039={TOOL_NO 5,BASE_NO 3,IPO_FRAME #BASE,POINT2[] " "}
DECL PDAT PP_OLP55={VEL 100.0,ACC 100.0,APO_DIST 100.0,APO_MODE #CDIS}
DECL E6POS Xl042={X -53.2410202,Y -294.750885,Z -178.516006,A -91.8654099,B -85.3020935,C 104.040001,S 2,T 35,E1 4299.97998,E2 0.0,E3 0.0,E4 0.0,E5 0.0,E6 0.0}
DECL FDAT Fl042={TOOL_NO 5,BASE_NO 3,IPO_FRAME #BASE,POINT2[] " "}
DECL E6POS XSWP_60_9171={X 191.517593,Y -817.554016,Z 112.109398,A -89.9988785,B 3.53138995,C 89.9993362,S 2,T 35,E1 4300.00195,E2 0.0,E3 0.0,E4 0.0,E5 0.0,E6 0.0}
DECL FDAT FSWP_60_9171={TOOL_NO 5,BASE_NO 3,IPO_FRAME #BASE,POINT2[] " ",TQ_STATE FALSE}
DECL E6POS XSWP_60_9173={X 190.195999,Y -817.508484,Z 58.3723106,A -89.9955215,B 25.9951591,C 90.0008163,S 2,T 35,E1 4299.98877,E2 0.0,E3 0.0,E4 0.0,E5 0.0,E6 0.0}
DECL FDAT FSWP_60_9173={TOOL_NO 5,BASE_NO 3,IPO_FRAME #BASE,POINT2[] " ",TQ_STATE FALSE}
DECL E6POS XSWP_60_9175={X 191.458801,Y -778.874573,Z 21.8832607,A -89.9954071,B 40.6308289,C 90.0165329,S 2,T 35,E1 4299.99805,E2 0.0,E3 0.0,E4 0.0,E5 0.0,E6 0.0}
DECL FDAT FSWP_60_9175={TOOL_NO 5,BASE_NO 3,IPO_FRAME #BASE,POINT2[] " ",TQ_STATE FALSE}
DECL E6POS XSWP_60_9177={X 192.126999,Y -741.065186,Z 23.4970093,A -89.9816132,B 80.5138321,C 90.019043,S 2,T 35,E1 4300.0,E2 0.0,E3 0.0,E4 0.0,E5 0.0,E6 0.0}
DECL FDAT FSWP_60_9177={TOOL_NO 5,BASE_NO 3,IPO_FRAME #BASE,POINT2[] " ",TQ_STATE FALSE}
DECL E6POS XSWP_60_9181={X 190.141907,Y -645.375916,Z 21.0312405,A 89.6592331,B 89.2380524,C -90.3413162,S 2,T 35,E1 4299.99902,E2 0.0,E3 0.0,E4 0.0,E5 0.0,E6 0.0}
DECL FDAT FSWP_60_9181={TOOL_NO 5,BASE_NO 3,IPO_FRAME #BASE,POINT2[] " ",TQ_STATE FALSE}
DECL E6POS XSWP_60_9183={X 190.654404,Y -596.434326,Z 20.9701595,A 89.993103,B 63.1963692,C -90.0092773,S 2,T 35,E1 4299.99902,E2 0.0,E3 0.0,E4 0.0,E5 0.0,E6 0.0}
DECL FDAT FSWP_60_9183={TOOL_NO 5,BASE_NO 3,IPO_FRAME #BASE,POINT2[] " ",TQ_STATE FALSE}
DECL E6POS XSWP_60_9185={X 191.043701,Y -548.768311,Z 63.8096199,A 89.9858627,B 55.4986191,C -90.0110779,S 2,T 35,E1 4299.99805,E2 0.0,E3 0.0,E4 0.0,E5 0.0,E6 0.0}
DECL FDAT FSWP_60_9185={TOOL_NO 5,BASE_NO 3,IPO_FRAME #BASE,POINT2[] " ",TQ_STATE FALSE}
DECL PDAT PP_OLP56={VEL 100.0,ACC 100.0,APO_DIST 100.0,APO_MODE #CDIS}
DECL E6POS Xl101={X 176.396698,Y -173.5616,Z 239.795593,A -90.0033875,B -45.0011406,C 90.0047836,S 2,T 35,E1 4300.00098,E2 0.0,E3 0.0,E4 0.0,E5 0.0,E6 0.0}
DECL FDAT Fl101={TOOL_NO 5,BASE_NO 3,IPO_FRAME #BASE,POINT2[] " "}
DECL PDAT PP_OLP57={VEL 100.0,ACC 100.0,APO_DIST 100.0,APO_MODE #CDIS}
DECL E6POS Xl102={X 181.552505,Y -125.495003,Z 257.162506,A -89.9991913,B -43.6211891,C 89.9991989,S 2,T 35,E1 4300.00391,E2 0.0,E3 0.0,E4 0.0,E5 0.0,E6 0.0}
DECL FDAT Fl102={TOOL_NO 5,BASE_NO 3,IPO_FRAME #BASE,POINT2[] " "}
DECL E6POS XSWP_60_9089={X 168.245102,Y -12.5500898,Z -45.5669899,A 89.2536087,B 84.5853119,C -91.5467072,S 2,T 3,E1 4299.99219,E2 0.0,E3 0.0,E4 0.0,E5 0.0,E6 0.0}
DECL FDAT FSWP_60_9089={TOOL_NO 5,BASE_NO 3,IPO_FRAME #BASE,POINT2[] " ",TQ_STATE FALSE}
DECL E6POS XSWP_60_9091={X 166.2948,Y -59.2193794,Z -46.0812607,A 89.2500763,B 84.5846481,C -91.5499268,S 2,T 3,E1 4299.99121,E2 0.0,E3 0.0,E4 0.0,E5 0.0,E6 0.0}
DECL FDAT FSWP_60_9091={TOOL_NO 5,BASE_NO 3,IPO_FRAME #BASE,POINT2[] " ",TQ_STATE FALSE}
DECL E6POS XSWP_60_9095={X 169.7771,Y -176.959702,Z -46.7267113,A 89.2638397,B 84.5842972,C -91.5364685,S 2,T 3,E1 4299.98877,E2 0.0,E3 0.0,E4 0.0,E5 0.0,E6 0.0}
DECL FDAT FSWP_60_9095={TOOL_NO 5,BASE_NO 3,IPO_FRAME #BASE,POINT2[] " ",TQ_STATE FALSE}
DECL E6POS XSWP_60_9097={X 170.790298,Y -224.4422,Z -28.7135906,A 87.3456116,B 87.5840073,C -93.4503632,S 2,T 3,E1 4299.98682,E2 0.0,E3 0.0,E4 0.0,E5 0.0,E6 0.0}
DECL FDAT FSWP_60_9097={TOOL_NO 5,BASE_NO 3,IPO_FRAME #BASE,POINT2[] " ",TQ_STATE FALSE}
DECL E6POS XSWP_60_7107={X 170.503494,Y -253.975998,Z -31.3881702,A 87.3448105,B 87.5836334,C -93.4512177,S 2,T 3,E1 4299.98584,E2 0.0,E3 0.0,E4 0.0,E5 0.0,E6 0.0}
DECL FDAT FSWP_60_7107={TOOL_NO 5,BASE_NO 3,IPO_FRAME #BASE,POINT2[] " ",TQ_STATE FALSE}
DECL E6POS XSWP_60_7101={X 169.488297,Y -295.904297,Z -19.4584503,A -80.6868362,B 89.0242767,C 98.5218124,S 2,T 3,E1 4299.98682,E2 0.0,E3 0.0,E4 0.0,E5 0.0,E6 0.0}
DECL FDAT FSWP_60_7101={TOOL_NO 5,BASE_NO 3,IPO_FRAME #BASE,POINT2[] " ",TQ_STATE FALSE}
DECL E6POS XSWP_60_7115={X 171.168396,Y -277.024506,Z 3.26121211,A -88.0905914,B 82.6041336,C 91.1257706,S 2,T 3,E1 4299.98584,E2 0.0,E3 0.0,E4 0.0,E5 0.0,E6 0.0}
DECL FDAT FSWP_60_7115={TOOL_NO 5,BASE_NO 3,IPO_FRAME #BASE,POINT2[] " ",TQ_STATE FALSE}
DECL E6POS XSWP_60_9103={X 169.092896,Y -357.490112,Z 54.5366707,A -89.9977264,B -0.003349012,C 90.0028915,S 2,T 35,E1 4299.99121,E2 0.0,E3 0.0,E4 0.0,E5 0.0,E6 0.0}
DECL FDAT FSWP_60_9103={TOOL_NO 5,BASE_NO 3,IPO_FRAME #BASE,POINT2[] " ",TQ_STATE FALSE}
DECL E6POS XSWP_60_7117={X 172.061096,Y -344.352509,Z 17.1497192,A -89.0555878,B 46.2205391,C 90.2096329,S 2,T 3,E1 4299.98389,E2 0.0,E3 0.0,E4 0.0,E5 0.0,E6 0.0}
DECL FDAT FSWP_60_7117={TOOL_NO 5,BASE_NO 3,IPO_FRAME #BASE,POINT2[] " ",TQ_STATE FALSE}
DECL E6POS XSWP_60_9113={X 173.390594,Y -275.042786,Z -112.536903,A -92.0510864,B -85.2995682,C 104.0205,S 2,T 35,E1 4299.979,E2 0.0,E3 0.0,E4 0.0,E5 0.0,E6 0.0}
DECL FDAT FSWP_60_9113={TOOL_NO 5,BASE_NO 3,IPO_FRAME #BASE,POINT2[] " ",TQ_STATE FALSE}
DECL LDAT LL_OLP49={VEL 2.0,ACC 100.0,APO_DIST 0.0,APO_FAC 0.0,ORI_TYP #VAR,CIRC_TYP #BASE,JERK_FAC 50.0}
DECL E6POS XSWP_60_7119={X 175.809799,Y -357.503296,Z 47.9063492,A -89.9979172,B -0.000778076181,C 90.0029831,S 2,T 35,E1 4299.98584,E2 0.0,E3 0.0,E4 0.0,E5 0.0,E6 0.0}
DECL FDAT FSWP_60_7119={TOOL_NO 5,BASE_NO 3,IPO_FRAME #BASE,POINT2[] " ",TQ_STATE FALSE}
DECL E6POS XSWP_60_7145={X 176.391495,Y -201.067398,Z 296.510803,A -90.005043,B -45.0009193,C 90.0062485,S 2,T 35,E1 4300.0,E2 0.0,E3 0.0,E4 0.0,E5 0.0,E6 0.0}
DECL FDAT FSWP_60_7145={TOOL_NO 5,BASE_NO 3,IPO_FRAME #BASE,POINT2[] " ",TQ_STATE FALSE}
DECL LDAT LL_OLP50={VEL 2.0,ACC 100.0,APO_DIST 0.0,APO_FAC 0.0,ORI_TYP #VAR,CIRC_TYP #BASE,JERK_FAC 50.0}
DECL PDAT PP_OLP29={VEL 100.0,ACC 100.0,APO_DIST 100.0,APO_MODE #CDIS}
DECL E6POS Xl071={X 73.9980011,Y -296.309692,Z 79.4658813,A -90.0,B -25.0,C 90.0,S 2,T 35,E1 4300.0,E2 0.0,E3 0.0,E4 0.0,E5 0.0,E6 0.0}
DECL FDAT Fl071={TOOL_NO 5,BASE_NO 3,IPO_FRAME #BASE,POINT2[] " "}
DECL PDAT PP_OLP30={VEL 100.0,ACC 100.0,APO_DIST 100.0,APO_MODE #CDIS}
DECL E6POS Xl072={X 82.3577881,Y -251.416397,Z 66.7752838,A -86.8620834,B -0.216702402,C 90.662117,S 2,T 35,E1 4299.99121,E2 0.0,E3 0.0,E4 0.0,E5 0.0,E6 0.0}
DECL FDAT Fl072={TOOL_NO 5,BASE_NO 3,IPO_FRAME #BASE,POINT2[] " "}
DECL PDAT PP_OLP31={VEL 100.0,ACC 100.0,APO_DIST 100.0,APO_MODE #CDIS}
DECL E6POS Xl076={X 176.474106,Y -332.770386,Z 66.7434082,A -89.0821915,B -0.216351107,C 90.6608734,S 2,T 35,E1 4299.99121,E2 0.0,E3 0.0,E4 0.0,E5 0.0,E6 0.0}
DECL FDAT Fl076={TOOL_NO 5,BASE_NO 3,IPO_FRAME #BASE,POINT2[] " "}
DECL LDAT LL_OLP51={VEL 2.0,ACC 100.0,APO_DIST 0.0,APO_FAC 0.0,ORI_TYP #VAR,CIRC_TYP #BASE,JERK_FAC 50.0}
DECL E6POS XSWP_60_7120={X 169.094101,Y -357.471313,Z 47.9132805,A -89.9972305,B -0.00383762107,C 90.0026169,S 2,T 35,E1 4299.99121,E2 0.0,E3 0.0,E4 0.0,E5 0.0,E6 0.0}
DECL FDAT FSWP_60_7120={TOOL_NO 5,BASE_NO 3,IPO_FRAME #BASE,POINT2[] " ",TQ_STATE FALSE}
DECL PDAT PP_OLP32={VEL 100.0,ACC 100.0,APO_DIST 100.0,APO_MODE #CDIS}
DECL E6POS Xl081={X 177.080307,Y -320.852997,Z 73.9970016,A -90.0,B -3.01534087E-08,C 90.0,S 2,T 35,E1 4300.0,E2 0.0,E3 0.0,E4 0.0,E5 0.0,E6 0.0}
DECL FDAT Fl081={TOOL_NO 5,BASE_NO 3,IPO_FRAME #BASE,POINT2[] " "}
DECL PDAT PP_OLP33={VEL 100.0,ACC 100.0,APO_DIST 100.0,APO_MODE #CDIS}
DECL E6POS Xl086={X 174.526398,Y -312.003998,Z 147.546005,A -90.0,B -5.00010014,C 90.0,S 2,T 35,E1 4300.0,E2 0.0,E3 0.0,E4 0.0,E5 0.0,E6 0.0}
DECL FDAT Fl086={TOOL_NO 5,BASE_NO 3,IPO_FRAME #BASE,POINT2[] " "}
DECL LDAT LL_OLP14={VEL 2.0,ACC 100.0,APO_DIST 0.0,APO_FAC 0.0,ORI_TYP #VAR,CIRC_TYP #BASE,JERK_FAC 50.0}
DECL E6POS XSWP_60_7128={X 168.644196,Y -353.469086,Z 159.192795,A -91.2637634,B -4.81876516,C 90.1613235,S 2,T 35,E1 4300.00488,E2 0.0,E3 0.0,E4 0.0,E5 0.0,E6 0.0}
DECL FDAT FSWP_60_7128={TOOL_NO 5,BASE_NO 3,IPO_FRAME #BASE,POINT2[] " "}
DECL LDAT LL_OLP24={VEL 2.0,ACC 100.0,APO_DIST 0.0,APO_FAC 0.0,ORI_TYP #VAR,CIRC_TYP #BASE,JERK_FAC 50.0}
DECL E6POS XSWP_60_7130={X 170.543503,Y -351.142609,Z 187.325104,A -90.0603714,B -4.99114323,C 89.4538193,S 2,T 35,E1 4300.00586,E2 0.0,E3 0.0,E4 0.0,E5 0.0,E6 0.0}
DECL FDAT FSWP_60_7130={TOOL_NO 5,BASE_NO 3,IPO_FRAME #BASE,POINT2[] " "}
DECL LDAT LL_OLP25={VEL 2.0,ACC 100.0,APO_DIST 0.0,APO_FAC 0.0,ORI_TYP #VAR,CIRC_TYP #BASE,JERK_FAC 50.0}
DECL E6POS XSWP_60_7132={X 169.933304,Y -347.036102,Z 217.126297,A -90.0359726,B -10.2011003,C 89.7093506,S 2,T 35,E1 4299.9668,E2 0.0,E3 0.0,E4 0.0,E5 0.0,E6 0.0}
DECL FDAT FSWP_60_7132={TOOL_NO 5,BASE_NO 3,IPO_FRAME #BASE,POINT2[] " "}
DECL LDAT LL_OLP37={VEL 2.0,ACC 100.0,APO_DIST 0.0,APO_FAC 0.0,ORI_TYP #VAR,CIRC_TYP #BASE,JERK_FAC 50.0}
DECL E6POS XSWP_60_7134={X 169.499298,Y -336.745697,Z 244.646698,A -90.0203934,B -10.0957804,C 89.8580627,S 2,T 35,E1 4299.97607,E2 0.0,E3 0.0,E4 0.0,E5 0.0,E6 0.0}
DECL FDAT FSWP_60_7134={TOOL_NO 5,BASE_NO 3,IPO_FRAME #BASE,POINT2[] " "}
DECL LDAT LL_OLP38={VEL 2.0,ACC 100.0,APO_DIST 0.0,APO_FAC 0.0,ORI_TYP #VAR,CIRC_TYP #BASE,JERK_FAC 50.0}
DECL E6POS XSWP_60_7136={X 170.150406,Y -321.261108,Z 266.513397,A -90.0109711,B -17.1879597,C 89.9056702,S 2,T 35,E1 4299.98389,E2 0.0,E3 0.0,E4 0.0,E5 0.0,E6 0.0}
DECL FDAT FSWP_60_7136={TOOL_NO 5,BASE_NO 3,IPO_FRAME #BASE,POINT2[] " "}
DECL LDAT LL_OLP39={VEL 2.0,ACC 100.0,APO_DIST 0.0,APO_FAC 0.0,ORI_TYP #VAR,CIRC_TYP #BASE,JERK_FAC 50.0}
DECL E6POS XSWP_60_7140={X 170.005005,Y -276.423798,Z 293.276794,A -89.9994736,B -26.2854691,C 89.9691772,S 2,T 35,E1 4300.00293,E2 0.0,E3 0.0,E4 0.0,E5 0.0,E6 0.0}
DECL FDAT FSWP_60_7140={TOOL_NO 5,BASE_NO 3,IPO_FRAME #BASE,POINT2[] " "}
DECL LDAT LL_OLP40={VEL 2.0,ACC 100.0,APO_DIST 0.0,APO_FAC 0.0,ORI_TYP #VAR,CIRC_TYP #BASE,JERK_FAC 50.0}
DECL E6POS XSWP_60_7142={X 167.399094,Y -256.003601,Z 300.454895,A -89.9894714,B -41.54916,C 89.9695969,S 2,T 35,E1 4299.99805,E2 0.0,E3 0.0,E4 0.0,E5 0.0,E6 0.0}
DECL FDAT FSWP_60_7142={TOOL_NO 5,BASE_NO 3,IPO_FRAME #BASE,POINT2[] " ",TQ_STATE FALSE}
DECL LDAT LL_OLP52={VEL 2.0,ACC 100.0,APO_DIST 0.0,APO_FAC 0.0,ORI_TYP #VAR,CIRC_TYP #BASE,JERK_FAC 50.0}
DECL E6POS XSWP_60_7144={X 169.806198,Y -237.515106,Z 299.451813,A -90.0080414,B -44.9938316,C 90.0089111,S 2,T 35,E1 4300.0,E2 0.0,E3 0.0,E4 0.0,E5 0.0,E6 0.0}
DECL FDAT FSWP_60_7144={TOOL_NO 5,BASE_NO 3,IPO_FRAME #BASE,POINT2[] " "}
DECL LDAT LL_OLP53={VEL 2.0,ACC 100.0,APO_DIST 0.0,APO_FAC 0.0,ORI_TYP #VAR,CIRC_TYP #BASE,JERK_FAC 50.0}
DECL E6POS XSWP_60_7146={X 170.010605,Y -197.472397,Z 299.145905,A -90.009697,B -44.9873314,C 90.0102463,S 2,T 35,E1 4300.0,E2 0.0,E3 0.0,E4 0.0,E5 0.0,E6 0.0}
DECL FDAT FSWP_60_7146={TOOL_NO 5,BASE_NO 3,IPO_FRAME #BASE,POINT2[] " ",TQ_STATE FALSE}
DECL PDAT PP_OLP58={VEL 100.0,ACC 100.0,APO_DIST 100.0,APO_MODE #CDIS}
DECL E6POS Xl103={X 169.240097,Y -207.901703,Z 267.68869,A -89.2902222,B -44.7676315,C 88.4695969,S 2,T 35,E1 4300.0,E2 0.0,E3 0.0,E4 0.0,E5 0.0,E6 0.0}
DECL FDAT Fl103={TOOL_NO 5,BASE_NO 3,IPO_FRAME #BASE,POINT2[] " "}
DECL PDAT PP_OLP59={VEL 100.0,ACC 100.0,APO_DIST 100.0,APO_MODE #CDIS}
DECL E6POS Xl104={X 172.770996,Y -80.8234177,Z 257.381012,A -89.5252075,B -29.7303295,C 88.3034363,S 2,T 35,E1 4300.00098,E2 0.0,E3 0.0,E4 0.0,E5 0.0,E6 0.0}
DECL FDAT Fl104={TOOL_NO 5,BASE_NO 3,IPO_FRAME #BASE,POINT2[] " "}
DECL LDAT LL_OLP54={VEL 2.0,ACC 100.0,APO_DIST 0.0,APO_FAC 0.0,ORI_TYP #VAR,CIRC_TYP #BASE,JERK_FAC 50.0}
DECL E6POS XSWP_60_7154={X 169.319504,Y -128.332901,Z 300.206207,A -90.0372009,B -36.5032387,C 90.023407,S 2,T 35,E1 4300.0,E2 0.0,E3 0.0,E4 0.0,E5 0.0,E6 0.0}
DECL FDAT FSWP_60_7154={TOOL_NO 5,BASE_NO 3,IPO_FRAME #BASE,POINT2[] " "}
DECL LDAT LL_OLP55={VEL 2.0,ACC 100.0,APO_DIST 0.0,APO_FAC 0.0,ORI_TYP #VAR,CIRC_TYP #BASE,JERK_FAC 50.0}
DECL E6POS XSWP_60_7156={X 170.647095,Y -36.9482384,Z 300.799103,A -90.0022278,B -29.9919109,C 90.0040512,S 2,T 35,E1 4300.00391,E2 0.0,E3 0.0,E4 0.0,E5 0.0,E6 0.0}
DECL FDAT FSWP_60_7156={TOOL_NO 5,BASE_NO 3,IPO_FRAME #BASE,POINT2[] " "}
DECL LDAT LL_OLP56={VEL 2.0,ACC 100.0,APO_DIST 0.0,APO_FAC 0.0,ORI_TYP #VAR,CIRC_TYP #BASE,JERK_FAC 50.0}
DECL E6POS XSWP_60_7158={X 170.960007,Y -2.66582203,Z 300.113098,A -89.9998322,B -29.9919395,C 90.0010834,S 2,T 35,E1 4300.00195,E2 0.0,E3 0.0,E4 0.0,E5 0.0,E6 0.0}
DECL FDAT FSWP_60_7158={TOOL_NO 5,BASE_NO 3,IPO_FRAME #BASE,POINT2[] " "}
DECL PDAT PP_OLP35={VEL 100.0,ACC 100.0,APO_DIST 100.0,APO_MODE #CDIS}
DECL E6POS Xl116={X 169.727005,Y -6.80677509,Z 253.825897,A -89.2291336,B -29.6888409,C 88.1471786,S 2,T 35,E1 4300.00195,E2 0.0,E3 0.0,E4 0.0,E5 0.0,E6 0.0}
DECL FDAT Fl116={TOOL_NO 5,BASE_NO 3,IPO_FRAME #BASE,POINT2[] " "}
DECL PDAT PP_OLP4={VEL 100.0,ACC 100.0,APO_DIST 100.0,APO_MODE #CDIS}
DECL E6POS Xl011={X 115.0243,Y -163.583496,Z 190.738495,A -89.5583496,B -79.2283707,C 90.2654724,S 2,T 35,E1 4299.99414,E2 0.0,E3 0.0,E4 0.0,E5 0.0,E6 0.0}
DECL FDAT Fl011={TOOL_NO 5,BASE_NO 3,IPO_FRAME #BASE,POINT2[] " "}
DECL PDAT PP_OLP45={VEL 100.0,ACC 100.0,APO_DIST 100.0,APO_MODE #CDIS}
DECL E6POS Xl015={X 187.548294,Y -200.192505,Z 48.43787,A 91.7383575,B 52.382061,C -90.1605988,S 2,T 3,E1 4299.99023,E2 0.0,E3 0.0,E4 0.0,E5 0.0,E6 0.0}
DECL FDAT Fl015={TOOL_NO 5,BASE_NO 3,IPO_FRAME #BASE,POINT2[] " "}
DECL LDAT LL_OLP57={VEL 2.0,ACC 100.0,APO_DIST 0.0,APO_FAC 0.0,ORI_TYP #VAR,CIRC_TYP #BASE,JERK_FAC 50.0}
DECL E6POS XSWP_60_9090={X 166.4655,Y -12.5319996,Z -45.5594482,A 89.247139,B 84.5920105,C -91.5547485,S 2,T 3,E1 4299.99414,E2 0.0,E3 0.0,E4 0.0,E5 0.0,E6 0.0}
DECL FDAT FSWP_60_9090={TOOL_NO 5,BASE_NO 3,IPO_FRAME #BASE,POINT2[] " ",TQ_STATE FALSE}
DECL LDAT LL_OLP58={VEL 2.0,ACC 100.0,APO_DIST 0.0,APO_FAC 0.0,ORI_TYP #VAR,CIRC_TYP #BASE,JERK_FAC 50.0}
DECL E6POS XSWP_60_9092={X 166.2948,Y -59.2193794,Z -46.0812607,A 89.2500763,B 84.5846481,C -91.5499268,S 2,T 3,E1 4299.99121,E2 0.0,E3 0.0,E4 0.0,E5 0.0,E6 0.0}
DECL FDAT FSWP_60_9092={TOOL_NO 5,BASE_NO 3,IPO_FRAME #BASE,POINT2[] " ",TQ_STATE FALSE}
DECL LDAT LL_OLP59={VEL 2.0,ACC 100.0,APO_DIST 0.0,APO_FAC 0.0,ORI_TYP #VAR,CIRC_TYP #BASE,JERK_FAC 50.0}
DECL E6POS XSWP_60_9151={X 167.267303,Y -103.972397,Z -46.4912605,A 89.2762527,B 84.5920868,C -91.5210876,S 2,T 3,E1 4299.99219,E2 0.0,E3 0.0,E4 0.0,E5 0.0,E6 0.0}
DECL FDAT FSWP_60_9151={TOOL_NO 5,BASE_NO 3,IPO_FRAME #BASE,POINT2[] " "}
DECL LDAT LL_OLP60={VEL 2.0,ACC 100.0,APO_DIST 0.0,APO_FAC 0.0,ORI_TYP #VAR,CIRC_TYP #BASE,JERK_FAC 50.0}
DECL E6POS XSWP_60_9096={X 167.694199,Y -177.091599,Z -46.7227516,A 89.2544479,B 84.5932922,C -91.5413284,S 2,T 3,E1 4299.98779,E2 0.0,E3 0.0,E4 0.0,E5 0.0,E6 0.0}
DECL FDAT FSWP_60_9096={TOOL_NO 5,BASE_NO 3,IPO_FRAME #BASE,POINT2[] " ",TQ_STATE FALSE}
DECL LDAT LL_OLP61={VEL 2.0,ACC 100.0,APO_DIST 0.0,APO_FAC 0.0,ORI_TYP #VAR,CIRC_TYP #BASE,JERK_FAC 50.0}
DECL E6POS XSWP_60_9098={X 168.227905,Y -224.578796,Z -28.7343597,A 87.3735504,B 87.5756836,C -93.4185715,S 2,T 3,E1 4299.98877,E2 0.0,E3 0.0,E4 0.0,E5 0.0,E6 0.0}
DECL FDAT FSWP_60_9098={TOOL_NO 5,BASE_NO 3,IPO_FRAME #BASE,POINT2[] " ",TQ_STATE FALSE}
DECL LDAT LL_OLP62={VEL 2.0,ACC 100.0,APO_DIST 0.0,APO_FAC 0.0,ORI_TYP #VAR,CIRC_TYP #BASE,JERK_FAC 50.0}
DECL E6POS XSWP_60_7108={X 169.062805,Y -253.955307,Z -31.5082798,A 87.4344864,B 87.5914078,C -93.3620071,S 2,T 3,E1 4299.98682,E2 0.0,E3 0.0,E4 0.0,E5 0.0,E6 0.0}
DECL FDAT FSWP_60_7108={TOOL_NO 5,BASE_NO 3,IPO_FRAME #BASE,POINT2[] " ",TQ_STATE FALSE}
DECL LDAT LL_OLP63={VEL 2.0,ACC 100.0,APO_DIST 0.0,APO_FAC 0.0,ORI_TYP #VAR,CIRC_TYP #BASE,JERK_FAC 50.0}
DECL E6POS XSWP_60_7102={X 169.488297,Y -295.904297,Z -19.4584503,A -80.6868362,B 89.0242767,C 98.5218124,S 2,T 3,E1 4299.98682,E2 0.0,E3 0.0,E4 0.0,E5 0.0,E6 0.0}
DECL FDAT FSWP_60_7102={TOOL_NO 5,BASE_NO 3,IPO_FRAME #BASE,POINT2[] " ",TQ_STATE FALSE}
DECL LDAT LL_OLP64={VEL 2.0,ACC 100.0,APO_DIST 0.0,APO_FAC 0.0,ORI_TYP #VAR,CIRC_TYP #BASE,JERK_FAC 50.0}
DECL E6POS XSWP_60_7116={X 171.168396,Y -277.024506,Z 3.26121211,A -88.0905914,B 82.6041336,C 91.1257706,S 2,T 3,E1 4299.98584,E2 0.0,E3 0.0,E4 0.0,E5 0.0,E6 0.0}
DECL FDAT FSWP_60_7116={TOOL_NO 5,BASE_NO 3,IPO_FRAME #BASE,POINT2[] " ",TQ_STATE FALSE}
DECL LDAT LL_OLP65={VEL 2.0,ACC 100.0,APO_DIST 0.0,APO_FAC 0.0,ORI_TYP #VAR,CIRC_TYP #BASE,JERK_FAC 50.0}
DECL E6POS XSWP_60_9104={X 171.724594,Y -316.937286,Z 3.99869704,A -88.8935471,B 65.3713684,C 90.3454819,S 2,T 3,E1 4299.99121,E2 0.0,E3 0.0,E4 0.0,E5 0.0,E6 0.0}
DECL FDAT FSWP_60_9104={TOOL_NO 5,BASE_NO 3,IPO_FRAME #BASE,POINT2[] " ",TQ_STATE FALSE}
DECL LDAT LL_OLP66={VEL 2.0,ACC 100.0,APO_DIST 0.0,APO_FAC 0.0,ORI_TYP #VAR,CIRC_TYP #BASE,JERK_FAC 50.0}
DECL E6POS XSWP_60_7118={X 168.248199,Y -347.425812,Z 21.3010502,A -89.0610504,B 46.2098503,C 90.2020264,S 2,T 3,E1 4299.98877,E2 0.0,E3 0.0,E4 0.0,E5 0.0,E6 0.0}
DECL FDAT FSWP_60_7118={TOOL_NO 5,BASE_NO 3,IPO_FRAME #BASE,POINT2[] " ",TQ_STATE FALSE}
DECL PDAT PP_OLP60={VEL 100.0,ACC 100.0,APO_DIST 100.0,APO_MODE #CDIS}
DECL E6POS Xl036={X 168.900604,Y -271.340607,Z 76.1519394,A -89.0555725,B 46.2203903,C 90.2092438,S 2,T 3,E1 4299.98389,E2 0.0,E3 0.0,E4 0.0,E5 0.0,E6 0.0}
DECL FDAT Fl036={TOOL_NO 5,BASE_NO 3,IPO_FRAME #BASE,POINT2[] " "}
DECL PDAT PP_OLP61={VEL 100.0,ACC 100.0,APO_DIST 100.0,APO_MODE #CDIS}
DECL E6POS Xl040={X 14.1120396,Y -278.348694,Z 74.4917068,A -89.0556335,B 46.2204819,C 90.2092819,S 2,T 3,E1 4299.98291,E2 0.0,E3 0.0,E4 0.0,E5 0.0,E6 0.0}
DECL FDAT Fl040={TOOL_NO 5,BASE_NO 3,IPO_FRAME #BASE,POINT2[] " "}
DECL PDAT PP_OLP62={VEL 100.0,ACC 100.0,APO_DIST 100.0,APO_MODE #CDIS}
DECL E6POS Xl043={X 31.9833298,Y -202.207504,Z 159.895203,A -88.5181198,B -65.9205627,C 94.9122467,S 2,T 35,E1 4299.98779,E2 0.0,E3 0.0,E4 0.0,E5 0.0,E6 0.0}
DECL FDAT Fl043={TOOL_NO 5,BASE_NO 3,IPO_FRAME #BASE,POINT2[] " "}
DECL PDAT PP_OLP63={VEL 100.0,ACC 100.0,APO_DIST 10.0,APO_MODE #CDIS}
DECL E6POS Xl044={X 31.9832306,Y -202.207504,Z 159.895096,A -88.5181198,B -65.9205627,C 94.9122391,S 2,T 35,E1 4299.98779,E2 0.0,E3 0.0,E4 0.0,E5 0.0,E6 0.0}
DECL FDAT Fl044={TOOL_NO 5,BASE_NO 3,IPO_FRAME #BASE,POINT2[] " "}
DECL E6POS XP1={X 201.0513,Y -814.501709,Z 57.3495293,A -89.8255692,B 25.9404907,C 89.9631577,S 2,T 35,E1 4299.98877,E2 0.0,E3 0.0,E4 0.0,E5 0.0,E6 0.0}
DECL FDAT FP1={TOOL_NO 5,BASE_NO 3,IPO_FRAME #BASE,POINT2[] " ",TQ_STATE FALSE}
DECL PDAT PPDAT1={VEL 100.0,ACC 100.0,APO_DIST 100.0}
DECL E6POS XP2={X 200.735901,Y -765.756104,Z 26.7770996,A -89.8061066,B 40.5903091,C 90.2168732,S 2,T 35,E1 4299.99805,E2 0.0,E3 0.0,E4 0.0,E5 0.0,E6 0.0}
DECL FDAT FP2={TOOL_NO 5,BASE_NO 3,IPO_FRAME #BASE,POINT2[] " ",TQ_STATE FALSE}
DECL PDAT PPDAT2={VEL 100.0,ACC 100.0,APO_DIST 100.0}
DECL E6POS XP3={X 205.502197,Y -596.439514,Z 20.9718304,A 89.993103,B 63.1963692,C -90.0092773,S 2,T 35,E1 4299.99902,E2 0.0,E3 0.0,E4 0.0,E5 0.0,E6 0.0}
DECL FDAT FP3={TOOL_NO 5,BASE_NO 3,IPO_FRAME #BASE,POINT2[] " ",TQ_STATE FALSE}
DECL PDAT PPDAT3={VEL 100.0,ACC 100.0,APO_DIST 100.0}
DECL E6POS XP4={X 201.262802,Y -551.140625,Z 63.8097115,A 89.9858627,B 55.4986191,C -90.0110779,S 2,T 35,E1 4299.99805,E2 0.0,E3 0.0,E4 0.0,E5 0.0,E6 0.0}
DECL FDAT FP4={TOOL_NO 5,BASE_NO 3,IPO_FRAME #BASE,POINT2[] " ",TQ_STATE FALSE}
DECL PDAT PPDAT4={VEL 100.0,ACC 100.0,APO_DIST 100.0}
DECL E6POS XP5={X 2793.50293,Y -5570.604,Z 775.185913,A 1.08841002,B -62.3716507,C 164.715302,S 2,T 3,E1 4299.98682,E2 0.0,E3 0.0,E4 0.0,E5 0.0,E6 0.0}
DECL FDAT FP5={TOOL_NO 6,BASE_NO 0,IPO_FRAME #BASE,POINT2[] " ",TQ_STATE FALSE}
DECL PDAT PPDAT5={VEL 100.0,ACC 100.0,APO_DIST 100.0,APO_MODE #CDIS}
DECL E6POS XP6={X 11.2346697,Y -260.635712,Z 168.615906,A 92.2102737,B -5.24029398,C -90.2750473,S 2,T 35,E1 4299.98193,E2 0.0,E3 0.0,E4 0.0,E5 0.0,E6 0.0}
DECL FDAT FP6={TOOL_NO 5,BASE_NO 3,IPO_FRAME #BASE,POINT2[] " ",TQ_STATE FALSE}
DECL PDAT PPDAT6={VEL 100.0,ACC 100.0,APO_DIST 100.0,APO_MODE #CDIS}
DECL PDAT Pvmax={VEL 100.0,ACC 100.0,APO_DIST 100.0}
DECL PDAT Pfin={VEL 100.0,ACC 100.0,APO_DIST 20.0,APO_MODE #CDIS}
DECL PDAT Psmall={VEL 100.0,ACC 100.0,APO_DIST 50.0,APO_MODE #CDIS}
DECL PDAT Plarge={VEL 100.0,ACC 100.0,APO_DIST 100.0,APO_MODE #CDIS}
DECL PDAT Pmedium={VEL 100.0,ACC 100.0,APO_DIST 100.0,APO_MODE #CDIS}
DECL PDAT Pxlarge={VEL 100.0,ACC 100.0,APO_DIST 500.0,APO_MODE #CDIS}
DECL E6POS XSWP_60_9117={X 168.644196,Y -353.469086,Z 159.192795,A -91.2637634,B -4.81876516,C 90.1613235,S 2,T 35,E1 4300.00488,E2 0.0,E3 0.0,E4 0.0,E5 0.0,E6 0.0}
DECL FDAT FSWP_60_9117={TOOL_NO 5,BASE_NO 3,IPO_FRAME #BASE,POINT2[] " ",TQ_STATE FALSE}
DECL E6POS XSWP_60_9119={X 170.543503,Y -351.142609,Z 187.325104,A -90.0603714,B -4.99114323,C 89.4538193,S 2,T 35,E1 4300.00586,E2 0.0,E3 0.0,E4 0.0,E5 0.0,E6 0.0}
DECL FDAT FSWP_60_9119={TOOL_NO 5,BASE_NO 3,IPO_FRAME #BASE,POINT2[] " ",TQ_STATE FALSE}
DECL E6POS XSWP_60_91129={X 169.933304,Y -347.036102,Z 217.126297,A -90.0359726,B -10.2011003,C 89.7093506,S 2,T 35,E1 4299.9668,E2 0.0,E3 0.0,E4 0.0,E5 0.0,E6 0.0}
DECL FDAT FSWP_60_91129={TOOL_NO 5,BASE_NO 3,IPO_FRAME #BASE,POINT2[] " ",TQ_STATE FALSE}
DECL E6POS XSWP_60_9121={X 169.933304,Y -347.036102,Z 217.126297,A -90.0359726,B -10.2011003,C 89.7093506,S 2,T 35,E1 4299.9668,E2 0.0,E3 0.0,E4 0.0,E5 0.0,E6 0.0}
DECL FDAT FSWP_60_9121={TOOL_NO 5,BASE_NO 3,IPO_FRAME #BASE,POINT2[] " ",TQ_STATE FALSE}
DECL E6POS XSWP_60_9123={X 169.499298,Y -336.745697,Z 244.646698,A -90.0203934,B -10.0957804,C 89.8580627,S 2,T 35,E1 4299.97607,E2 0.0,E3 0.0,E4 0.0,E5 0.0,E6 0.0}
DECL FDAT FSWP_60_9123={TOOL_NO 5,BASE_NO 3,IPO_FRAME #BASE,POINT2[] " ",TQ_STATE FALSE}
DECL E6POS XSWP_60_9125={X 170.150406,Y -321.261108,Z 266.513397,A -90.0109711,B -17.1879597,C 89.9056702,S 2,T 35,E1 4299.98389,E2 0.0,E3 0.0,E4 0.0,E5 0.0,E6 0.0}
DECL FDAT FSWP_60_9125={TOOL_NO 5,BASE_NO 3,IPO_FRAME #BASE,POINT2[] " ",TQ_STATE FALSE}
DECL E6POS XSWP_60_9129={X 170.005005,Y -276.423798,Z 293.276794,A -89.9932022,B -35.7904091,C 89.9659271,S 2,T 35,E1 4300.00293,E2 0.0,E3 0.0,E4 0.0,E5 0.0,E6 0.0}
DECL FDAT FSWP_60_9129={TOOL_NO 5,BASE_NO 3,IPO_FRAME #BASE,POINT2[] " ",TQ_STATE FALSE}
DECL E6POS XSWP_60_9131={X 167.398895,Y -257.46579,Z 300.561188,A -89.9894714,B -41.54916,C 89.9695969,S 2,T 35,E1 4299.99805,E2 0.0,E3 0.0,E4 0.0,E5 0.0,E6 0.0}
DECL FDAT FSWP_60_9131={TOOL_NO 5,BASE_NO 3,IPO_FRAME #BASE,POINT2[] " ",TQ_STATE FALSE}
DECL E6POS XSWP_60_9133={X 169.806198,Y -237.515106,Z 299.451813,A -90.0080414,B -44.9938316,C 90.0089111,S 2,T 35,E1 4300.0,E2 0.0,E3 0.0,E4 0.0,E5 0.0,E6 0.0}
DECL FDAT FSWP_60_9133={TOOL_NO 5,BASE_NO 3,IPO_FRAME #BASE,POINT2[] " ",TQ_STATE FALSE}
DECL E6POS XSWP_60_9135={X 170.010605,Y -197.472397,Z 299.145905,A -90.009697,B -44.9873314,C 90.0102463,S 2,T 35,E1 4300.0,E2 0.0,E3 0.0,E4 0.0,E5 0.0,E6 0.0}
DECL FDAT FSWP_60_9135={TOOL_NO 5,BASE_NO 3,IPO_FRAME #BASE,POINT2[] " ",TQ_STATE FALSE}
DECL E6POS XSWP_60_7159={X 170.194794,Y -69.7142029,Z 299.795197,A -90.0021362,B -30.0117893,C 90.0030365,S 2,T 35,E1 4300.00098,E2 0.0,E3 0.0,E4 0.0,E5 0.0,E6 0.0}
DECL FDAT FSWP_60_7159={TOOL_NO 5,BASE_NO 3,IPO_FRAME #BASE,POINT2[] " "}
DECL E6POS XSWP_60_9137={X 168.023499,Y -157.253906,Z 299.967712,A -90.036972,B -40.6139793,C 90.0259171,S 2,T 35,E1 4300.0,E2 0.0,E3 0.0,E4 0.0,E5 0.0,E6 0.0}
DECL FDAT FSWP_60_9137={TOOL_NO 5,BASE_NO 3,IPO_FRAME #BASE,POINT2[] " ",TQ_STATE FALSE}
DECL E6POS XSWP_60_9139={X 169.317902,Y -128.331299,Z 300.209808,A -90.0371933,B -36.503231,C 90.0235138,S 2,T 35,E1 4300.0,E2 0.0,E3 0.0,E4 0.0,E5 0.0,E6 0.0}
DECL FDAT FSWP_60_9139={TOOL_NO 5,BASE_NO 3,IPO_FRAME #BASE,POINT2[] " ",TQ_STATE FALSE}
DECL E6POS XSWP_60_9140={X 170.779205,Y -65.7698822,Z 301.053986,A -90.0324326,B -32.1959991,C 90.0185013,S 2,T 35,E1 4300.00195,E2 0.0,E3 0.0,E4 0.0,E5 0.0,E6 0.0}
DECL FDAT FSWP_60_9140={TOOL_NO 5,BASE_NO 3,IPO_FRAME #BASE,POINT2[] " ",TQ_STATE FALSE}
DECL E6POS XSWP_60_9143={X 170.778397,Y -65.7698364,Z 301.052185,A -90.0324631,B -32.1964607,C 90.0185471,S 2,T 35,E1 4300.00098,E2 0.0,E3 0.0,E4 0.0,E5 0.0,E6 0.0}
DECL FDAT FSWP_60_9143={TOOL_NO 5,BASE_NO 3,IPO_FRAME #BASE,POINT2[] " ",TQ_STATE FALSE}
DECL E6POS XSWP_60_9145={X 170.647095,Y -36.9482384,Z 300.799103,A -90.0022278,B -29.9919109,C 90.0040512,S 2,T 35,E1 4300.00391,E2 0.0,E3 0.0,E4 0.0,E5 0.0,E6 0.0}
DECL FDAT FSWP_60_9145={TOOL_NO 5,BASE_NO 3,IPO_FRAME #BASE,POINT2[] " ",TQ_STATE FALSE}
DECL E6POS XSWP_60_9147={X 170.960007,Y -2.66582203,Z 300.113098,A -89.9998322,B -29.9919395,C 90.0010834,S 2,T 35,E1 4300.00195,E2 0.0,E3 0.0,E4 0.0,E5 0.0,E6 0.0}
DECL FDAT FSWP_60_9147={TOOL_NO 5,BASE_NO 3,IPO_FRAME #BASE,POINT2[] " ",TQ_STATE FALSE}
DECL E6POS XSWP_60_9041={X 192.730392,Y -882.800476,Z -187.645203,A -89.9909134,B -79.9946594,C 89.9927597,S 2,T 35,E1 4300.00195,E2 0.0,E3 0.0,E4 0.0,E5 0.0,E6 0.0}
DECL FDAT FSWP_60_9041={TOOL_NO 5,BASE_NO 3,IPO_FRAME #BASE,POINT2[] " ",TQ_STATE FALSE}
DECL E6POS XSWP_60_9039={X 192.190796,Y -853.006714,Z -159.147797,A -89.9849777,B -79.9993362,C 89.9846191,S 2,T 35,E1 4300.00781,E2 0.0,E3 0.0,E4 0.0,E5 0.0,E6 0.0}
DECL FDAT FSWP_60_9039={TOOL_NO 5,BASE_NO 3,IPO_FRAME #BASE,POINT2[] " ",TQ_STATE FALSE}
DECL E6POS XSWP_60_9037={X 192.047394,Y -824.388977,Z -130.335602,A -90.0232315,B -79.9922714,C 90.0233917,S 2,T 35,E1 4300.00781,E2 0.0,E3 0.0,E4 0.0,E5 0.0,E6 0.0}
DECL FDAT FSWP_60_9037={TOOL_NO 5,BASE_NO 3,IPO_FRAME #BASE,POINT2[] " ",TQ_STATE FALSE}
DECL E6POS XSWP_60_9035={X 192.727097,Y -795.518616,Z -101.527298,A -90.0249176,B -79.9941635,C 90.024353,S 2,T 35,E1 4299.979,E2 0.0,E3 0.0,E4 0.0,E5 0.0,E6 0.0}
DECL FDAT FSWP_60_9035={TOOL_NO 5,BASE_NO 3,IPO_FRAME #BASE,POINT2[] " ",TQ_STATE FALSE}
DECL E6POS XSWP_60_9033={X 190.991699,Y -769.520874,Z -74.9092331,A -90.0168304,B -80.0018311,C 90.0171814,S 2,T 35,E1 4299.98682,E2 0.0,E3 0.0,E4 0.0,E5 0.0,E6 0.0}
DECL FDAT FSWP_60_9033={TOOL_NO 5,BASE_NO 3,IPO_FRAME #BASE,POINT2[] " ",TQ_STATE FALSE}
DECL E6POS XSWP_60_9029={X 191.9142,Y -697.815674,Z -49.9122505,A 90.0055695,B -65.0068436,C -89.9991074,S 2,T 35,E1 4300.03076,E2 0.0,E3 0.0,E4 0.0,E5 0.0,E6 0.0}
DECL FDAT FSWP_60_9029={TOOL_NO 5,BASE_NO 3,IPO_FRAME #BASE,POINT2[] " ",TQ_STATE FALSE}
DECL E6POS XSWP_60_9027={X 190.732803,Y -659.745789,Z -55.9621696,A 89.9975815,B -65.006691,C -89.9963226,S 2,T 35,E1 4300.00293,E2 0.0,E3 0.0,E4 0.0,E5 0.0,E6 0.0}
DECL FDAT FSWP_60_9027={TOOL_NO 5,BASE_NO 3,IPO_FRAME #BASE,POINT2[] " ",TQ_STATE FALSE}
DECL E6POS XSWP_60_9025={X 193.292206,Y -623.187927,Z -72.8630524,A 90.0108032,B -65.0110321,C -90.0050583,S 2,T 35,E1 4299.9541,E2 0.0,E3 0.0,E4 0.0,E5 0.0,E6 0.0}
DECL FDAT FSWP_60_9025={TOOL_NO 5,BASE_NO 3,IPO_FRAME #BASE,POINT2[] " ",TQ_STATE FALSE}
DECL E6POS XSWP_60_9023={X 193.7789,Y -600.831482,Z -92.8529663,A 90.0178909,B -65.0057373,C -90.0168228,S 2,T 35,E1 4300.01611,E2 0.0,E3 0.0,E4 0.0,E5 0.0,E6 0.0}
DECL FDAT FSWP_60_9023={TOOL_NO 5,BASE_NO 3,IPO_FRAME #BASE,POINT2[] " ",TQ_STATE FALSE}
DECL E6POS XP7={X 201.262802,Y -551.140625,Z 63.8097115,A 89.9858627,B 55.4986191,C -90.0110779,S 2,T 35,E1 4299.99805,E2 0.0,E3 0.0,E4 0.0,E5 0.0,E6 0.0}
DECL FDAT FP7={TOOL_NO 5,BASE_NO 3,IPO_FRAME #BASE,POINT2[] " ",TQ_STATE FALSE}
DECL E6POS Xl077={X 171.776001,Y -268.065613,Z 267.479889,A -89.3132706,B -41.3269501,C 88.4377823,S 2,T 35,E1 4299.99805,E2 0.0,E3 0.0,E4 0.0,E5 0.0,E6 0.0}
DECL FDAT Fl077={TOOL_NO 5,BASE_NO 3,IPO_FRAME #BASE,POINT2[] " "}
DECL E6POS Xl078={X 171.824005,Y -201.652802,Z 267.515198,A -89.3133316,B -41.3269997,C 88.4377136,S 2,T 35,E1 4299.99707,E2 0.0,E3 0.0,E4 0.0,E5 0.0,E6 0.0}
DECL FDAT Fl078={TOOL_NO 5,BASE_NO 3,IPO_FRAME #BASE,POINT2[] " "}
ENDDAT
